// TIA Portal V16 program export: 5 tag tables, 16 data types, 1 data blocks, 21 code blocks (in call order from the OBs), 0 instance data blocks

VAR_GLOBAL   // PLC tag table "Default tag table"
END_VAR

VAR_GLOBAL   // PLC tag table "GLOBAL_CONSTANTS"
END_VAR
VAR_GLOBAL CONSTANT   // user constants
   NUM_AI_RACK : UInt := 1;   // Number of physical analog input points used per rack.
   NUM_DQ_RACK : UInt := 4;   // Number of physical digital output points used per rack.
   NUM_DQ_ROOM : UInt := 9;   // Number of physical digital output points used per room.
   MAX_DQ_PER_ROOM : UInt := 40;   // Max number of physical digital output points per room-based IO module. This needs to equal (NUM_DQ_ROOM + NUM_DQ_RACK*MAX_RACKS_PER_ROOM + EXTRA_DQ_PER_ROOM).
   MAX_VFDS : UInt := 6;   // Total number of VFDs configured in the HW config. This needs to equal MAX_ROOMS * MAX_RACKS_PER_ROOM.
   MAX_ROOMS : UInt := 1;   // Maximum possible number of rooms controlled by a given PLC
   MAX_RACKS_PER_ROOM : UInt := 6;   // Maximum possible number of racks per room
   NUM_AI_ROOM : UInt := 13;   // Number of physical analog input points used per room.
   EXTRA_DQ_PER_ROOM : UInt := 7;   // Number of unused physical digital output points per room-based IO module.
   EXTRA_AI_PER_ROOM : UInt := 1;   // Number of unused physical analog input points per room-based IO module.
   MAX_AI_PER_ROOM : UInt := 20;   // Max number of physical analog input points per room-based IO module. This needs to equal (NUM_AI_ROOM + NUM_AI_RACK*MAX_RACKS_PER_ROOM + EXTRA_AI_PER_ROOM).
END_VAR

VAR_GLOBAL   // PLC tag table "IO"
   GlobalAI AT %I100.0 : "udtArrAIGlobal";   //    {ExternalAccessible false, ExternalVisible false, ExternalWritable false}
   GlobalDQ AT %Q100.0 : "udtArrDQGlobal";   //    {ExternalAccessible false, ExternalVisible false, ExternalWritable false}
END_VAR

VAR_GLOBAL   // PLC tag table "Library Constants"
END_VAR
VAR_GLOBAL CONSTANT   // user constants
   eSTATE_MANUAL : Int := 2;   // State Machine enumeration
   ePBLT_FLASHING_ENABLED : Int := 4;   // HMI PB LT enumeration
   eSTATE_RETRACTING : Int := 5;   // State Machine enumeration
   "IoScaling.S7Analog.Ni100.rScaledMax" : Real := 250.0;
   "IoScaling.S7Analog.Ni100.Climate.rScaledMax" : Real := 250.0;
   eSTEP_StoppingStart : Int := 4000;   // State Machine enumeration
   eSTEP_VerifyCenterComplete : Int := 7999;   // State Machine enumeration
   "IoScaling.S7Analog.150Ohms.rScaledMax" : Real := 150.0;
   "IoScaling.S7Analog.Default.bSwapBytes" : Bool := false;
   eANALOG_INPUTHIGHHIGH : Int := 102;
   eMOTION_DISABLED : Int := 4;   // Status Enumeration - Motion
   "IoScaling.S7Analog.Pt100.iRawMax" : Int := 8500;
   eSTEP_RetractingComplete : Int := 5999;   // State Machine enumeration
   eMODE_MANUAL : Int := 2;   // Mode enumeration
   eANALOG_INPUTINVALID : Int := 101;
   ePBLT_HIDDEN : Int := -1;   // HMI PB LT enumeration
   eVALVE_HOMEON : Int := 6;
   "IoScaling.S7Analog.Pt100.Climate.rScaledMin" : Real := -120.0;
   eHOME_ABS_RET_ABS : Int := 7;   // See MC_Home help for details
   eMOTION_ERROR : Int := 0;   // Status Enumeration - Motion
   ePB_MAINTAINED : Int := 1;   // HMI PB Type enumeration
   LKINCTRL_LENGTH_OF_PATHDATA_NAME : Int := 10;
   LKINCTRL_NO_OF_PATHDATA_ELEMENTS : Int := 15;
   "IoScaling.S7Analog.Pt100.Climate.iRawMax" : Int := 13000;
   eVALVE_ERROR : Int := 2;
   "IoScaling.S7Analog.Types.Pt100.Climate" : Int := 3;
   eMODE_INDEPENDENT : Int := 10;   // Mode
   "IoScaling.S7Analog.600Ohms.rScaledMax" : Real := 600.0;
   eMOTION_RUNNING : Int := 2;   // Status Enumeration - Motion
   "IoScaling.S7Analog.Ni100.Climate.rScaledMin" : Real := -60.0;
   eMOTION_STOPPED : Int := 1;   // Status Enumeration - Motion
   eMOTION_MAINTENANCE : Int := 3;   // Status Enumeration - Motion
   "IoScaling.S7Analog.Ni100.rScaledMin" : Real := -60.0;
   eSTATE_STOPPING : Int := 4;   // State Machine enumeration
   "IoScaling.S7Analog.Pt100.Climate.rScaledMax" : Real := 130.0;
   "IoScaling.S7Analog.Pt100.rScaledMax" : Real := 850.0;
   "IoScaling.S7Analog.Types.Ni100.Climate" : Int := 5;
   ePB_UNLATCH : Int := 3;   // HMI PB Type enumeration
   "IoScaling.S7Analog.Ni100.Climate.iRawMax" : Int := 25000;
   eSTEP_BladeChangeStart : Int := 6000;   // State Machine enumeration
   "IoScaling.S7Analog.300Ohms.rScaledMin" : Real := 0.0;
   "IoScaling.S7Analog.Types.Pt100" : Int := 2;
   LKINCTRL_PI : LReal := 3.1415926535897932846264;
   eVALVE_WORKPOSITION : Int := 3;
   eCAM_SYNCDIRECTION_SHORTESTWAY : Int := 3;   // See MC_CamIn help for details
   "IoScaling.S7Analog.Types.+-V/mA" : Int := 1;
   ePBLT_FLASHING_DISABLED : Int := 5;   // HMI PB LT enumeration
   "IoScaling.S7Analog.150Ohms.rScaledMin" : Real := 0.0;
   eHOME_ACCEPT_CURRENT : Int := 11;   // Used when the configured and current encoders don't match
   LKINCTRL_NO_OF_START_EXECUTE_CMDS : Int := 5;
   ePBLT_TRANSITIONING : Int := 2;   // HMI PB LT enumeration
   SM_ACTIVE_DYNAMICS : Int := 0;
   eVALVE_WORKON : Int := 5;
   "IoScaling.S7Analog.+-V/mA.iRawMax" : Int := 27648;
   eSTATE_INITIALIZATION : Int := 1;   // State Machine enumeration
   LKINCTRL_NO_OF_PATHDATA_PREBUFFER_ELEMENTS : Int := 5;
   eHOME_ABS_RET_OFFSET : Int := 6;   // See MC_Home help for details
   eSTEP_BladeChangeComplete : Int := 6999;   // State Machine enumeration
   eSTEP_RunningComplete : Int := 3999;   // State Machine enumeration
   eANALOG_READY : Int := 100;
   ePBLT_ENABLED : Int := 1;   // HMI PB LT enumeration
   "IoScaling.S7Analog.Pt100.Climate.iRawMin" : Int := -12000;
   eSTATE_RUNNING : Int := 3;   // State Machine enumeration
   LKINCTRL_NO_OF_LAST_FLAG : Int := 15;
   "IoScaling.S7Analog.Ni100.iRawMax" : Int := 2500;
   "IoScaling.S7Analog.Types.Default" : Int := 0;
   eHOME_ACCEPT_CONFIG : Int := 12;   // Used when the configured and current encoders don't match
   eSTEP_RunningStart : Int := 3000;   // State Machine enumeration
   "IoScaling.S7Analog.Default.iRawMin" : Int := 0;
   ePBLT_ACTIVE : Int := 3;   // HMI PB LT enumeration
   "IoScaling.S7Analog.Types.Ni100" : Int := 4;
   eMODE_AUTO : Int := 1;   // Mode enumeration
   "IoScaling.S7Analog.Default.iRawMax" : Int := 27648;
   ePBLT_DISABLED : Int := 0;   // HMI PB LT enumeration
   LKINCTRL_NO_OF_SEQ_EXECUTE_CMDS : Int := 5;
   eSTEP_StoppingComplete : Int := 4999;   // State Machine enumeration
   "IoScaling.S7Analog.Ni100.Climate.iRawMin" : Int := -6000;
   "IoScaling.S7Analog.Pt100.iRawMin" : Int := -2000;
   ePB_LATCH : Int := 2;   // HMI PB Type enumeration
   eVALVE_ESTOP : Int := 1;
   eSTEP_RetractingStart : Int := 5000;   // State Machine enumeration
   "IoScaling.S7Analog.300Ohms.rScaledMax" : Real := 300.0;
   eANALOG_INPUTLOW : Int := 105;
   "IoScaling.S7Analog.Pt100.rScaledMin" : Real := -200.0;
   eSTATE_BLADECHANGE : Int := 6;   // State Machine enumeration
   "IoScaling.S7Analog.600Ohms.rScaledMin" : Real := 0.0;
   eSTATE_VERIFYCENTER : Int := 7;   // State Machine enumeration
   eVALVE_STOPPED : Int := 0;
   eCAM_SYNCPROFILEREFERENCE_LEADINGVALUEDISTANCE : Int := 1;   // See MC_CamIn help for details
   "IoScaling.S7Analog.Ni100.iRawMin" : Int := -600;
   ePB_HELD : Int := 4;   // HMI PB Type enumeration
   LKINCTRL_NO_OF_CMD_SETFLAGS : Int := 8;
   eSTEP_VerifyCenterStart : Int := 7000;   // State Machine enumeration
   eVALVE_HOMEPOSITION : Int := 4;
   eANALOG_INPUTHIGH : Int := 104;
   eANALOG_INPUTLOWLOW : Int := 103;
   "IoScaling.S7Analog.+-V/mA.iRawMin" : Int := -27648;
   ePB_MOMENTARY : Int := 0;   // HMI PB Type enumeration
   "Modes.PID.Pretuning" : Int := 1;
   "TotalizerTimeUnits.DAYS" : Int := 4;
   "HMI.Status.ForwardWork" : Int := 3;
   "FIFO.iQueueDisabled" : Int := -1;
   "Handshakes.iSize" : Int := 5;
   "Modes.Auto" : Int := 1;
   "HMI.Status.Generic1" : Int := 101;
   "Simocode.Types.DirectStarter" : Int := 1;
   "Estop.MinSetPoint" : Int := 0;
   "Simocode.Types.OverloadRelay" : Int := 0;
   "HMI.Status.SimulatedReverseHome" : Int := 8;
   "TotalizerTimeUnits.MILLISECONDS" : Int := 0;
   "HMI.Status.Generic4" : Int := 104;
   "SoftStarter.HMI.Status.EStop" : Int := 1;
   "HMI.Status.OnForwardWork" : Int := 5;
   "DataTypes.iMaxInt" : Int := 32767;
   "FIFO.iQueueSize" : Int := 5;
   "Modes.PID.ManualMode" : Int := 4;
   "TotalizerTimeUnits.SECONDS" : Int := 1;
   "SoftStarter.Types.3RW30" : Int := 30;
   "HMI.Status.Generic3" : Int := 103;
   "HMI.Status.OnReverseHome" : Int := 6;
   "HMI.Status.Estop" : Int := 1;
   "SoftStarter.HMI.Status.Error" : Int := 2;
   "HMI.Status.Generic6" : Int := 106;
   "DataTypes.rMaxReal" : Real := 3.402823e38;
   "SoftStarter.HMI.Status.Off" : Int := 0;
   "Modes.PID.Inactive" : Int := 0;
   "HMI.Status.GenericNone" : Int := 100;
   "HMI.Status.Generic2" : Int := 102;
   "Modes.PID.AutoMode" : Int := 3;
   "SoftStarter.HMI.Status.On" : Int := 4;
   "Estop.HMISetPoint" : Int := 2;
   "HMI.Status.ReverseHome" : Int := 4;
   "DataTypes.rMinReal" : Real := -3.402823e38;
   "TotalizerTimeUnits.MINUTES" : Int := 2;
   "Modes.PID.FineTuning" : Int := 2;
   "TotalizerTimeUnits.HOURS" : Int := 3;
   "Ramp.Timed" : Int := 1;
   "Estop.MaxSetPoint" : Int := 1;
   "SoftStarter.Types.3RW40" : Int := 40;
   "Ramp.Continuous" : Int := 0;
   "HMI.Status.Generic5" : Int := 105;
   "Modes.Manual" : Int := 2;
   "Modes.Stop" : Int := 0;
   "HMI.Status.SimulatedOnReverseHome" : Int := 10;
   "Simocode.Types.ReversingStarter" : Int := 2;
   "Modes.Independent" : Int := 10;
   "DataTypes.iMinInt" : Int := -32768;
   "SoftStarter.HMI.Status.RampUp" : Int := 3;
   "SoftStarter.HMI.Status.RampDown" : Int := 5;
   "HMI.Status.Error" : Int := 2;
   "HMI.Status.SimulatedOnForwardWork" : Int := 9;
   "HMI.Status.SimulatedForwardWork" : Int := 7;
   "HMI.Status.Stopped" : Int := 0;
END_VAR

VAR_GLOBAL   // PLC tag table "System Bits"
   System_Byte AT %MB1 : Byte;   //    {ExternalAccessible false, ExternalVisible false, ExternalWritable false}
   AlwaysFALSE AT %M1.3 : Bool;   //    {ExternalAccessible false, ExternalVisible false, ExternalWritable false}
   "Clock_1.25Hz" AT %M0.4 : Bool;   //    {ExternalAccessible false, ExternalVisible false, ExternalWritable false}
   Clock_1Hz AT %M0.5 : Bool;   //    {ExternalAccessible false, ExternalVisible false, ExternalWritable false}
   "Clock_0.5Hz" AT %M0.7 : Bool;   //    {ExternalAccessible false, ExternalVisible false, ExternalWritable false}
   FirstScan AT %M1.0 : Bool;   //    {ExternalAccessible false, ExternalVisible false, ExternalWritable false}
   Clock_Byte AT %MB0 : Byte;   //    {ExternalAccessible false, ExternalVisible false, ExternalWritable false}
   "Clock_2.5Hz" AT %M0.2 : Bool;   //    {ExternalAccessible false, ExternalVisible false, ExternalWritable false}
   "Clock_0.625Hz" AT %M0.6 : Bool;   //    {ExternalAccessible false, ExternalVisible false, ExternalWritable false}
   Clock_5Hz AT %M0.1 : Bool;   //    {ExternalAccessible false, ExternalVisible false, ExternalWritable false}
   Clock_10Hz AT %M0.0 : Bool;   //    {ExternalAccessible false, ExternalVisible false, ExternalWritable false}
   AlwaysTRUE AT %M1.2 : Bool;   //    {ExternalAccessible false, ExternalVisible false, ExternalWritable false}
   DiagStatusUpdate AT %M1.1 : Bool;   //    {ExternalAccessible false, ExternalVisible false, ExternalWritable false}
   Clock_2Hz AT %M0.3 : Bool;   //    {ExternalAccessible false, ExternalVisible false, ExternalWritable false}
END_VAR

TYPE "udtFertigationSettings"
VERSION : 0.1
   STRUCT
      tMeasurementTime { ExternalAccessible := 'False'; ExternalVisible := 'False'; ExternalWritable := 'False'} : Time;   // Duration of cycle through M loop before measurement taken (s)
      rMeasurementVolume { ExternalAccessible := 'False'; ExternalVisible := 'False'; ExternalWritable := 'False'} : Real;   // Amount of water to receive from rack for measurement (L)
      bNutrientAEnable { ExternalAccessible := 'False'; ExternalVisible := 'False'; ExternalWritable := 'False'} : Bool;   // Enables nutrient A for use in dosing
      bNutrientBEnable { ExternalAccessible := 'False'; ExternalVisible := 'False'; ExternalWritable := 'False'} : Bool;   // Enables nutrient B for use in dosing
      rISELowSP { ExternalAccessible := 'False'; ExternalVisible := 'False'; ExternalWritable := 'False'} : Real;   // Low setpoint for ISE measurement for dosing
      rISEHighSP { ExternalAccessible := 'False'; ExternalVisible := 'False'; ExternalWritable := 'False'} : Real;   // High setpoint for ISE measurement for dosing
      tNutrientDosingDuration { ExternalAccessible := 'False'; ExternalVisible := 'False'; ExternalWritable := 'False'} : Time;   // Duration for which to add a nutrient during dosing (s)
      bDosingActive { ExternalAccessible := 'False'; ExternalVisible := 'False'; ExternalWritable := 'False'} : Bool;   // Rack was dosed on last MD cycle and is below high SP
      rOperatingVolume { ExternalAccessible := 'False'; ExternalVisible := 'False'; ExternalWritable := 'False'} : Real;   // Operating volume for fill after dosing (L)
      rTotalShelfVolume { ExternalAccessible := 'False'; ExternalVisible := 'False'; ExternalWritable := 'False'} : Real;
      rMaxReservoirVolume { ExternalAccessible := 'False'; ExternalVisible := 'False'; ExternalWritable := 'False'} : Real;   // Maximum water capacity of the rack (L)
      rMinReservoirVolume { ExternalAccessible := 'False'; ExternalVisible := 'False'; ExternalWritable := 'False'} : Real;   // Minimum water capacity of the rack (L)
      rRackCurrentVolume { ExternalAccessible := 'False'; ExternalVisible := 'False'; ExternalWritable := 'False'} : Real;   // Current rack fill level (L)
      bPumpAtStandstill { ExternalAccessible := 'False'; ExternalVisible := 'False'; ExternalWritable := 'False'} : Bool;
      bEndDischargeCommand { ExternalAccessible := 'False'; ExternalVisible := 'False'; ExternalWritable := 'False'} : Bool;
      tDischargeTime { ExternalAccessible := 'False'; ExternalVisible := 'False'; ExternalWritable := 'False'} : Time;
      bEnableIncomingRotate { ExternalAccessible := 'False'; ExternalVisible := 'False'; ExternalWritable := 'False'} : Bool;   // Rack is in M&D mode and circulating state
   END_STRUCT;

END_TYPE

TYPE "udtModbusValBool"
VERSION : 0.1
   STRUCT
      iAddr { ExternalAccessible := 'False'; ExternalVisible := 'False'; ExternalWritable := 'False'} : UInt;   // Full modbus address (1 indexed, including offset for object type)
      bVal { ExternalAccessible := 'False'; ExternalVisible := 'False'; ExternalWritable := 'False'} : Bool;
   END_STRUCT;

END_TYPE

TYPE "udtModbusValReal"
VERSION : 0.1
   STRUCT
      iRegister { ExternalAccessible := 'False'; ExternalVisible := 'False'; ExternalWritable := 'False'} : UInt;   // Full modbus address (1 indexed, including offset for object type)
      rVal { ExternalAccessible := 'False'; ExternalVisible := 'False'; ExternalWritable := 'False'} : Real;
   END_STRUCT;

END_TYPE

TYPE "udtNutrientReading"
VERSION : 0.1
   STRUCT
      rISEReading { ExternalVisible := 'False'; ExternalWritable := 'False'} : Real;   // Nutrient measurement level
      rORPReading { ExternalVisible := 'False'; ExternalWritable := 'False'} : Real;   // Nutrient measurement level
      rECReading { ExternalVisible := 'False'; ExternalWritable := 'False'} : Real;   // Nutrient measurement level
      rpHReading { ExternalVisible := 'False'; ExternalWritable := 'False'} : Real;   // Nutrient measurement level
   END_STRUCT;

END_TYPE

TYPE "udtTimeOfDaySetpoint"
VERSION : 0.1
   STRUCT
      TimeOfDaySeconds { ExternalVisible := 'False'} : DInt := -1;   // -1 default for unused setpoint
      rSetpoint { ExternalVisible := 'False'} : Real;
   END_STRUCT;

END_TYPE

TYPE "udtArrAIGlobal"
VERSION : 0.1
   STRUCT
      Room { ExternalAccessible := 'False'; ExternalVisible := 'False'; ExternalWritable := 'False'; S7_SetPoint := 'False'} : Array[1.."MAX_ROOMS"] of "udtArrAIRoom";
   END_STRUCT;

END_TYPE

TYPE "udtArrAIRoom"
VERSION : 0.1
   STRUCT
      AI { ExternalAccessible := 'False'; ExternalVisible := 'False'; ExternalWritable := 'False'} : Array[1.."MAX_AI_PER_ROOM"] of Int;
   END_STRUCT;

END_TYPE

TYPE "udtArrDQGlobal"
VERSION : 0.1
   STRUCT
      Room { ExternalAccessible := 'False'; ExternalVisible := 'False'; ExternalWritable := 'False'; S7_SetPoint := 'False'} : Array[1.."MAX_ROOMS"] of "udtArrDQRoom";
   END_STRUCT;

END_TYPE

TYPE "udtArrDQRoom"
VERSION : 0.1
   STRUCT
      DQ { ExternalAccessible := 'False'; ExternalVisible := 'False'; ExternalWritable := 'False'} : Array[1.."MAX_DQ_PER_ROOM"] of Bool;
   END_STRUCT;

END_TYPE

TYPE "udtDigitalOutput"
VERSION : 0.1
   STRUCT
      bAutoVal { ExternalVisible := 'False'; ExternalWritable := 'False'} : Bool;   // Value set by the program
      bOverrideVal { ExternalVisible := 'False'} : Bool;   // Value set by the user, tracks bAuto when bOverrideEnable=0
      bStatus { ExternalVisible := 'False'; ExternalWritable := 'False'} : Bool;   // Value being written to actual output
      bOverrideEnable { ExternalVisible := 'False'} : Bool;   // Sets bOut to bOverride
   END_STRUCT;

END_TYPE

TYPE "udtRackAI"
VERSION : 0.1
   STRUCT
      IW_ReservoirLevel { ExternalAccessible := 'False'; ExternalVisible := 'False'; ExternalWritable := 'False'} : Int;
   END_STRUCT;

END_TYPE

TYPE "udtRackDQ"
VERSION : 0.1
   STRUCT
      Q_SupplySolenoid { ExternalAccessible := 'False'; ExternalVisible := 'False'; ExternalWritable := 'False'} : Bool;
      Q_ReturnSolenoid { ExternalAccessible := 'False'; ExternalVisible := 'False'; ExternalWritable := 'False'} : Bool;
      Q_ShelfSolenoid { ExternalAccessible := 'False'; ExternalVisible := 'False'; ExternalWritable := 'False'} : Bool;
      Q_Lights { ExternalAccessible := 'False'; ExternalVisible := 'False'; ExternalWritable := 'False'} : Bool;
   END_STRUCT;

END_TYPE

TYPE "udtRoomAI"
VERSION : 0.1
   STRUCT
      IW_RoomTemperature_1 { ExternalAccessible := 'False'; ExternalVisible := 'False'; ExternalWritable := 'False'} : Int;
      IW_RoomTemperature_2 { ExternalAccessible := 'False'; ExternalVisible := 'False'; ExternalWritable := 'False'} : Int;
      IW_RoomHumidity_1 { ExternalAccessible := 'False'; ExternalVisible := 'False'; ExternalWritable := 'False'} : Int;
      IW_RoomHumidity_2 { ExternalAccessible := 'False'; ExternalVisible := 'False'; ExternalWritable := 'False'} : Int;
      IW_TankLevel { ExternalAccessible := 'False'; ExternalVisible := 'False'; ExternalWritable := 'False'} : Int;
      IW_NutrientALevel { ExternalAccessible := 'False'; ExternalVisible := 'False'; ExternalWritable := 'False'} : Int;
      IW_NutrientBLevel { ExternalAccessible := 'False'; ExternalVisible := 'False'; ExternalWritable := 'False'} : Int;
      IW_NutrientAcidLevel { ExternalAccessible := 'False'; ExternalVisible := 'False'; ExternalWritable := 'False'} : Int;
      IW_pHSensor { ExternalAccessible := 'False'; ExternalVisible := 'False'; ExternalWritable := 'False'} : Int;
      IW_ECSensor { ExternalAccessible := 'False'; ExternalVisible := 'False'; ExternalWritable := 'False'} : Int;
      IW_ISESensor { ExternalAccessible := 'False'; ExternalVisible := 'False'; ExternalWritable := 'False'} : Int;
      IW_ORPSensor { ExternalAccessible := 'False'; ExternalVisible := 'False'; ExternalWritable := 'False'} : Int;
      IW_CO2Sensor { ExternalAccessible := 'False'; ExternalVisible := 'False'; ExternalWritable := 'False'} : Int;
   END_STRUCT;

END_TYPE

TYPE "udtRoomDQ"
VERSION : 0.1
   STRUCT
      Q_MPathSolenoid { ExternalAccessible := 'False'; ExternalVisible := 'False'; ExternalWritable := 'False'} : Bool;
      Q_FreshWaterSolenoid { ExternalAccessible := 'False'; ExternalVisible := 'False'; ExternalWritable := 'False'} : Bool;
      Q_DischargeSolenoid { ExternalAccessible := 'False'; ExternalVisible := 'False'; ExternalWritable := 'False'} : Bool;
      Q_TankReturnSolenoid { ExternalAccessible := 'False'; ExternalVisible := 'False'; ExternalWritable := 'False'} : Bool;
      Q_NutrientAEnable { ExternalAccessible := 'False'; ExternalVisible := 'False'; ExternalWritable := 'False'} : Bool;
      Q_NutrientBEnable { ExternalAccessible := 'False'; ExternalVisible := 'False'; ExternalWritable := 'False'} : Bool;
      Q_NutrientAcidEnable { ExternalAccessible := 'False'; ExternalVisible := 'False'; ExternalWritable := 'False'} : Bool;
      Q_NutrientMixingPumps { ExternalAccessible := 'False'; ExternalVisible := 'False'; ExternalWritable := 'False'} : Bool;
      Q_CO2Solenoid { ExternalAccessible := 'False'; ExternalVisible := 'False'; ExternalWritable := 'False'} : Bool;
   END_STRUCT;

END_TYPE

TYPE "udtError_VFD"
VERSION : 0.1
   STRUCT
      MotorProtectorTripped { ExternalWritable := 'False'} : Bool;   // Motor protector tripped
      LocalDisconnectOff { ExternalWritable := 'False'} : Bool;   // Motor disconnect off
      ClutchTripped { ExternalWritable := 'False'} : Bool;   // Clutch tripped
      NoContactorFeedback { ExternalWritable := 'False'} : Bool;   // No feedback from motor contactor
      ContactorStillOn { ExternalWritable := 'False'} : Bool;   // Contactor still on
      NoSignalForward { ExternalWritable := 'False'} : Bool;   // No signal forward from VFD
      NoSignalReverse { ExternalWritable := 'False'} : Bool;   // No signal reverse from VFD
      MotorNotStopped { ExternalWritable := 'False'} : Bool;   // Motor doesn't stop
      MaxFrequencyReached { ExternalWritable := 'False'} : Bool;   // Max frequency reached
      Overcurrent { ExternalWritable := 'False'} : Bool;   // VFD overcurrent
      MotorOverload { ExternalWritable := 'False'} : Bool;   // Motor overload
      VFDOverload { ExternalWritable := 'False'} : Bool;   // VFD overload
      GeneralFault { ExternalWritable := 'False'} : Bool;   // VFD fault
      NoCoolingFanFeedback { ExternalWritable := 'False'} : Bool;   // No feedback from cooling fan
   END_STRUCT;

END_TYPE

TYPE "udtHMI_VFD_Control"
VERSION : 0.1
   STRUCT
      iMode : Int;   // Current mode
      iErrorCode { ExternalWritable := 'False'} : Int;   // Error code
      iStatus { ExternalWritable := 'False'} : Int;   // Status for HMI display
      rManualSpeedSP { S7_SetPoint := 'True'} : Real;   // Speed set point for manual mode
      rAutoSpeedSP { ExternalWritable := 'False'} : Real;   // Speed set point for automatic mode
      rActualSpeed { ExternalWritable := 'False'} : Real;   // Actual motor speed
      rActualCurrent { ExternalWritable := 'False'} : Real;   // Actual motor current
      rActualPower { ExternalWritable := 'False'} : Real;   // Actual motor power
      bPB_ResetError : Bool;   // PB Reset errors
      bPB_Forward : Bool;   // PB Move forward in manual mode
      bPB_Reverse : Bool;   // PB Move reverse in manual mode
      bPB_Stop : Bool;   // PB Stop in manual mode
      bPBEN_ResetError { ExternalWritable := 'False'} : Bool;   // PB Reset errors enabled
      bPBEN_Forward { ExternalWritable := 'False'} : Bool;   // PB Forward enabled
      bPBEN_Reverse { ExternalWritable := 'False'} : Bool;   // PB Reverse enabled
      bPBEN_Stop { ExternalWritable := 'False'} : Bool;   // PB Stop enabled
      bForwardOn { ExternalWritable := 'False'} : Bool;   // Moving forward
      bReverseOn { ExternalWritable := 'False'} : Bool;   // Moving Reverse
      bSignalForward { ExternalWritable := 'False'} : Bool;   // Forward signal
      bSignalReverse { ExternalWritable := 'False'} : Bool;   // Reverse signal
      bError { ExternalWritable := 'False'} : Bool;   // Overall error
      bInterlock { ExternalWritable := 'False'} : Bool;   // VFD Interlocked
   END_STRUCT;

END_TYPE

DATA_BLOCK "dbMain"
{ S7_Optimized_Access := 'TRUE' }
VERSION : 0.1
NON_RETAIN
"fbMain"

BEGIN
   Room[1].Fertigation.Controls.rTankEmptyLevel := 60.0;
   Room[1].AI_ISESensor.Config.rHighCalibration := 900.0;

END_DATA_BLOCK

ORGANIZATION_BLOCK "Main"   // OB1, LAD, ProgramCycle
TITLE = "Main Program Sweep (Cycle)"
{ S7_Optimized_Access := 'TRUE' }
VERSION : 0.1
// stored: AutoNumber true, IsIECCheckEnabled false, SetENOAutomatically false
   VAR_INPUT
      Initial_Call : Bool;   // Initial call of this OB
      Remanence : Bool;   // =True, if remanent data are available
   END_VAR
BEGIN

REGION Network 1
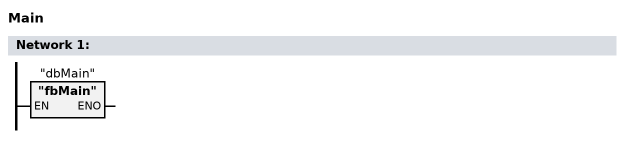
   RUNG wire#powerrail
      "dbMain"()
   END_RUNG
   // the same network as SCL:
   "dbMain"();   // "fbMain"
END_REGION
END_ORGANIZATION_BLOCK

FUNCTION_BLOCK "fbMain"   // FB4, LAD
{ S7_Optimized_Access := 'TRUE' }
VERSION : 0.1
// Main block which calls all room FBs and holds all parameters in instance memory.
// stored: AutoNumber true, IsIECCheckEnabled false, IsRetainMemResEnabled false, MemoryReserve 100, SetENOAutomatically false, UDAEnableTagReadback false
   VAR
      Room { ExternalVisible := 'False'} : Array[1.."MAX_ROOMS"] of "fbRoom";
      Config { ExternalVisible := 'False'} : "fbConfig";
   END_VAR
   VAR_TEMP
      iRoomCount : Int;
      iRackCount : Int;
      iPos : DInt;
   END_VAR
BEGIN

REGION Network 1 (SCL): Call config FB
   // bInSimulation := TRUE skips IO device configuration steps
   #Config(bInSimulation := #Config.bInSimulation);
END_REGION

REGION Network 2 (SCL): Map input array to all room and rack inputs
   IF #Config.Status.bDone THEN

       FOR #iRoomCount := 1 TO UINT_TO_INT("MAX_ROOMS") DO

           #iPos := 1; // input array is 1 indexed

           MOVE_BLK(IN := "GlobalAI".Room[#iRoomCount].AI[#iPos],
                    COUNT := "NUM_AI_ROOM",
                    OUT => #Room[#iRoomCount].arrAI[1]);

           #iPos += "NUM_AI_ROOM";


           FOR #iRackCount := 1 TO UINT_TO_INT("MAX_RACKS_PER_ROOM") DO

               MOVE_BLK(IN := "GlobalAI".Room[#iRoomCount].AI[#iPos],
                        COUNT := "NUM_AI_RACK",
                        OUT => #Room[#iRoomCount].Rack[#iRackCount].arrAI[1]);

               #iPos += "NUM_AI_RACK";

           END_FOR;

           #iPos += "EXTRA_AI_PER_ROOM"; // skip over unused points

       END_FOR;

   END_IF;
END_REGION

REGION Network 3 (SCL): TEMPORARY- Remap inputs from temporary IO tag table
   #Room[1].arrAI[1] := "IW_RoomTemperature_1";
   #Room[1].arrAI[2] := "IW_RoomTemperature_2";
   #Room[1].arrAI[3] := "IW_RoomHumidity_1";
   #Room[1].arrAI[4] := "IW_RoomHumidity_2";
   #Room[1].arrAI[5] := "IW_TankLevel";
   #Room[1].arrAI[6] := "IW_NutrientALevel";
   #Room[1].arrAI[7] := "IW_NutrientBLevel";
   #Room[1].arrAI[8] := "IW_NutrientAcidLevel";
   #Room[1].arrAI[9] := "IW_pHSensor";
   #Room[1].arrAI[10] := "IW_ECSensor";
   #Room[1].arrAI[11] := "IW_ISESensor";
   #Room[1].arrAI[12] := "IW_ORPSensor";
   #Room[1].arrAI[13] := "IW_CO2Sensor";

   #Room[1].Rack[1].arrAI[1] := "IW_Rack1Level";
   #Room[1].Rack[2].arrAI[1] := "IW_Rack2Level";
   #Room[1].Rack[3].arrAI[1] := "IW_Rack3Level";
   #Room[1].Rack[4].arrAI[1] := "IW_Rack4Level";
   #Room[1].Rack[5].arrAI[1] := "IW_Rack5Level";
   #Room[1].Rack[6].arrAI[1] := "IW_Rack6Level";
END_REGION

REGION Network 4 (SCL): Call FBs for all configured rooms
   IF #Config.Status.bDone THEN

       FOR #iRoomCount := 1 TO #Config.iNumRooms DO

           #Room[#iRoomCount](arrAI := #Room[#iRoomCount].arrAI,
                              arrDQ=> #Room[#iRoomCount].arrDQ);

       END_FOR;

   END_IF;
END_REGION

REGION Network 5 (SCL): Combine all room and rack outputs into a single output array
   IF #Config.Status.bDone THEN

       FOR #iRoomCount := 1 TO UINT_TO_INT("MAX_ROOMS") DO

           #iPos := 1; // output array is 1 indexed

           MOVE_BLK(IN := #Room[#iRoomCount].arrDQ[1],
                    COUNT := "NUM_DQ_ROOM",
                    OUT => "GlobalDQ".Room[#iRoomCount].DQ[#iPos]);

           #iPos += "NUM_DQ_ROOM";


           FOR #iRackCount := 1 TO UINT_TO_INT("MAX_RACKS_PER_ROOM") DO

               MOVE_BLK(IN := #Room[#iRoomCount].Rack[#iRackCount].arrDQ[1],
                        COUNT := "NUM_DQ_RACK",
                        OUT => "GlobalDQ".Room[#iRoomCount].DQ[#iPos]);

               #iPos += "NUM_DQ_RACK";

           END_FOR;

           #iPos += "EXTRA_DQ_PER_ROOM"; // skip over unused points

       END_FOR;

   END_IF;
END_REGION

REGION Network 6 (SCL): TEMPORARY- Remap inputs to temporary IO tag table
   "Q_MPathSolenoid" := #Room[1].arrDQ[1];
   "Q_FreshWaterSolenoid" := #Room[1].arrDQ[2];
   "Q_DischargeSolenoid" := #Room[1].arrDQ[3];
   "Q_TankReturnSolenoid" := #Room[1].arrDQ[4];
   "Q_NutrientAEnable" := #Room[1].arrDQ[5];
   "Q_NutrientBEnable" := #Room[1].arrDQ[6];
   "Q_NutrientAcidEnable" := #Room[1].arrDQ[7];
   "Q_NutrientMixingPumps" := #Room[1].arrDQ[8];
   "Q_CO2Solenoid" := #Room[1].arrDQ[9];

   "Q_Rack1Supply" := #Room[1].Rack[1].arrDQ[1];
   "Q_Rack1Return" := #Room[1].Rack[1].arrDQ[2];
   "Q_Rack1Shelves" := #Room[1].Rack[1].arrDQ[3];
   "Q_Rack1Lights" := #Room[1].Rack[1].arrDQ[4];
   "Q_Rack2Supply" := #Room[1].Rack[2].arrDQ[1];
   "Q_Rack2Return" := #Room[1].Rack[2].arrDQ[2];
   "Q_Rack2Shelves" := #Room[1].Rack[2].arrDQ[3];
   "Q_Rack2Lights" := #Room[1].Rack[2].arrDQ[4];
   "Q_Rack3Supply" := #Room[1].Rack[3].arrDQ[1];
   "Q_Rack3Return" := #Room[1].Rack[3].arrDQ[2];
   "Q_Rack3Shelves" := #Room[1].Rack[3].arrDQ[3];
   "Q_Rack3Lights" := #Room[1].Rack[3].arrDQ[4];
   "Q_Rack4Supply" := #Room[1].Rack[4].arrDQ[1];
   "Q_Rack4Return" := #Room[1].Rack[4].arrDQ[2];
   "Q_Rack4Shelves" := #Room[1].Rack[4].arrDQ[3];
   "Q_Rack4Lights" := #Room[1].Rack[4].arrDQ[4];
   "Q_Rack5Supply" := #Room[1].Rack[5].arrDQ[1];
   "Q_Rack5Return" := #Room[1].Rack[5].arrDQ[2];
   "Q_Rack5Shelves" := #Room[1].Rack[5].arrDQ[3];
   "Q_Rack5Lights" := #Room[1].Rack[5].arrDQ[4];
   "Q_Rack6Supply" := #Room[1].Rack[6].arrDQ[1];
   "Q_Rack6Return" := #Room[1].Rack[6].arrDQ[2];
   "Q_Rack6Shelves" := #Room[1].Rack[6].arrDQ[3];
   "Q_Rack6Lights" := #Room[1].Rack[6].arrDQ[4];
END_REGION
END_FUNCTION_BLOCK

FUNCTION_BLOCK "fbConfig"
{ S7_Optimized_Access := 'TRUE' }
VERSION : 0.1
   VAR_INPUT RETAIN
      bInSimulation { ExternalAccessible := 'False'; ExternalVisible := 'False'; ExternalWritable := 'False'} : Bool := false;   // If true, skips IO reconfig steps
   END_VAR

   VAR RETAIN
      Controls { ExternalVisible := 'False'} : Struct
         iSetNumRooms { ExternalVisible := 'False'} : Int := 1;
         arrSetNumRacksPerRoom { ExternalVisible := 'False'} : Array[1.."MAX_ROOMS"] of Int := [6];
         bSetConfig { ExternalVisible := 'False'} : Bool := false;
      END_STRUCT;
   END_VAR
   VAR 
      Status { ExternalVisible := 'False'; ExternalWritable := 'False'} : Struct
         bDone { ExternalVisible := 'False'; ExternalWritable := 'False'} : Bool;
         bBusy { ExternalVisible := 'False'; ExternalWritable := 'False'} : Bool;
         bError { ExternalVisible := 'False'; ExternalWritable := 'False'} : Bool;
         ErrorMsg { ExternalVisible := 'False'; ExternalWritable := 'False'} : String;
      END_STRUCT;
      iNumRooms { ExternalVisible := 'False'; ExternalWritable := 'False'} : Int := 0;
      iStep { ExternalAccessible := 'False'; ExternalVisible := 'False'; ExternalWritable := 'False'} : Int;
      iNextStep { ExternalAccessible := 'False'; ExternalVisible := 'False'; ExternalWritable := 'False'} : Int;
      R_TRIG_SetConfig {InstructionName := 'R_TRIG'; LibVersion := '1.0'; ExternalAccessible := 'False'; ExternalVisible := 'False'; ExternalWritable := 'False'} : R_TRIG;
      ReconfigIOSystem {InstructionName := 'ReconfigIOSystem'; LibVersion := '1.2'; ExternalAccessible := 'False'; ExternalVisible := 'False'; ExternalWritable := 'False'; S7_SetPoint := 'False'} : ReconfigIOSystem;
      arrVfdDeviceConfig { ExternalAccessible := 'False'; ExternalVisible := 'False'; ExternalWritable := 'False'} : Array[-2.."MAX_VFDS"] of Word;
   END_VAR

   VAR_TEMP 
      iRoomIndex : Int;
      iRackIndex : Int;
      arrTelegrams : Array[1.."MAX_VFDS"] of HW_SUBMODULE;
      arrIoDeviceIds : Array[1.."MAX_VFDS"] of HW_DEVICE;
      i : Int;
      iVfdCount : Int;
      bSettingsValid : Bool;
      strErrorCode : String;
      retVal : Word;
   END_VAR

   VAR CONSTANT 
      eStep_ValidateConfig : Int;
      eStep_SetUp : Int := 1;
      eStep_Deactivate : Int := 2;
      eStep_WaitForDeactivate : Int := 3;
      eStep_Reconfig : Int := 4;
      eStep_WaitForReconfig : Int := 5;
      eStep_Restart : Int := 6;
      eStep_Done : Int := 7;
      eStep_Error : Int := 8;
   END_VAR


BEGIN
	// Enables VFDs and IO racks based on the number of configured rooms and racks.
	// The intention is for everything to be configurable via the OPC UA interface and nothing
	// needs to be changed in TIA Portal, so that all deployments regardless of size can use the same codebase.
	
	// Global constants for reference:
	(*
	"MAX_ROOMS"
	"MAX_RACKS_PER_ROOM"
	"MAX_VFDS"
	
	"NUM_AI_ROOM"
	"NUM_AI_RACK"
	"MAX_AI_TOTAL"
	
	"NUM_DQ_ROOM"
	"NUM_DQ_RACK"
	"MAX_DQ_TOTAL"
	*)
	
	REGION 0: Validate config, set num racks and rooms
	    
	    // wait for start command
	    #R_TRIG_SetConfig(CLK:= #Controls.bSetConfig);
	    
	    // also trigger on PLC startup
	    IF "FirstScan" OR #iStep = #eStep_ValidateConfig OR
	        (#R_TRIG_SetConfig.Q AND (#iStep = #eStep_Done OR #iStep = #eStep_Error) ) THEN
	        
	        REGION Check error conditions            
	            // make sure specified number of rooms and racks is valid
	            #bSettingsValid := TRUE;
	            #Status.ErrorMsg := '';
	            
	            IF "MAX_VFDS" <> "MAX_ROOMS" * "MAX_RACKS_PER_ROOM" THEN
	                #bSettingsValid := FALSE;
	                #Status.ErrorMsg := CONCAT(IN1 := #Status.ErrorMsg, IN2 := ' MAX_VFDS != MAX_ROOMS*MAX_RACKS ');
	            END_IF;
	            
	            IF #Controls.iSetNumRooms > "MAX_ROOMS" THEN
	                #bSettingsValid := FALSE;
	                #Status.ErrorMsg := CONCAT(IN1 := #Status.ErrorMsg, IN2 := ' NumRooms > MAX ');
	            END_IF;
	            
	            FOR #i := 1 TO UINT_TO_INT("MAX_ROOMS") DO
	                IF #Controls.arrSetNumRacksPerRoom[#i] > "MAX_RACKS_PER_ROOM" THEN
	                    #bSettingsValid := FALSE;
	                    #Status.ErrorMsg := CONCAT(IN1 := #Status.ErrorMsg, IN2 := ' NumRacks > MAX ');
	                    EXIT;
	                END_IF;
	            END_FOR;
	            
	            IF "MAX_AI_PER_ROOM" <> ("NUM_AI_ROOM" + "NUM_AI_RACK" * "MAX_RACKS_PER_ROOM" + "EXTRA_AI_PER_ROOM") OR ( "MAX_AI_PER_ROOM" MOD 4 <> 0) THEN
	                #bSettingsValid := FALSE;
	                #Status.ErrorMsg := CONCAT(IN1 := #Status.ErrorMsg, IN2 := ' MAX_AI_PER_ROOM incorrect ');
	            END_IF;
	            
	            IF "MAX_DQ_PER_ROOM" <> ("NUM_DQ_ROOM" + "NUM_DQ_RACK" * "MAX_RACKS_PER_ROOM" + "EXTRA_DQ_PER_ROOM") OR ( "MAX_DQ_PER_ROOM" MOD 8 <> 0) THEN
	                #bSettingsValid := FALSE;
	                #Status.ErrorMsg := CONCAT(IN1 := #Status.ErrorMsg, IN2 := ' MAX_DQ_PER_ROOM incorrect ');
	            END_IF;
	            
	        END_REGION
	        
	        IF #bSettingsValid THEN
	            // set number of rooms
	            #iNumRooms := #Controls.iSetNumRooms;
	            
	            FOR #iRoomIndex := 1 TO #iNumRooms DO
	                // set number of racks in each room
	                "dbMain".Room[#iRoomIndex].Config.iNumRacks := #Controls.arrSetNumRacksPerRoom[#iRoomIndex];
	            END_FOR;
	            
	            #iNextStep := #eStep_SetUp;
	            
	        ELSE
	            #iNextStep := #eStep_Error;
	            
	        END_IF;
	        
	    END_IF;
	    
	END_REGION
	
	REGION 1: Set up params
	    
	    IF #iStep = #eStep_SetUp THEN
	        
	        REGION Map VFD IO device system constants
	            // Populate temp array of system constants for all possible VFDs
	            #arrIoDeviceIds[1] := "RackPumpVFD_1~PROFINET_interface~IODevice";
	            #arrIoDeviceIds[2] := "RackPumpVFD_2~PROFINET_interface~IODevice";
	            #arrIoDeviceIds[3] := "RackPumpVFD_3~PROFINET_interface~IODevice";
	            #arrIoDeviceIds[4] := "RackPumpVFD_4~PROFINET_interface~IODevice";
	            #arrIoDeviceIds[5] := "RackPumpVFD_5~PROFINET_interface~IODevice";
	            #arrIoDeviceIds[6] := "RackPumpVFD_6~PROFINET_interface~IODevice";
	            (*
	            #arrIoDeviceIds[7] := "RackPumpVFD_7~PROFINET_interface~IODevice";
	            #arrIoDeviceIds[8] := "RackPumpVFD_8~PROFINET_interface~IODevice";
	            #arrIoDeviceIds[9] := "RackPumpVFD_9~PROFINET_interface~IODevice";
	            #arrIoDeviceIds[10] := "RackPumpVFD_10~PROFINET_interface~IODevice";
	            #arrIoDeviceIds[11] := "RackPumpVFD_11~PROFINET_interface~IODevice";
	            #arrIoDeviceIds[12] := "RackPumpVFD_12~PROFINET_interface~IODevice";
	            
	            
	            #arrIoDeviceIds[13] := "RackPumpVFD_13~PROFINET_interface~IODevice";
	            #arrIoDeviceIds[14] := "RackPumpVFD_14~PROFINET_interface~IODevice";
	            #arrIoDeviceIds[15] := "RackPumpVFD_15~PROFINET_interface~IODevice";
	            #arrIoDeviceIds[16] := "RackPumpVFD_16~PROFINET_interface~IODevice";
	            #arrIoDeviceIds[17] := "RackPumpVFD_17~PROFINET_interface~IODevice";
	            #arrIoDeviceIds[18] := "RackPumpVFD_18~PROFINET_interface~IODevice";
	            #arrIoDeviceIds[19] := "RackPumpVFD_19~PROFINET_interface~IODevice";
	            #arrIoDeviceIds[20] := "RackPumpVFD_20~PROFINET_interface~IODevice";
	            #arrIoDeviceIds[21] := "RackPumpVFD_21~PROFINET_interface~IODevice";
	            #arrIoDeviceIds[22] := "RackPumpVFD_22~PROFINET_interface~IODevice";
	            #arrIoDeviceIds[23] := "RackPumpVFD_23~PROFINET_interface~IODevice";
	            #arrIoDeviceIds[24] := "RackPumpVFD_24~PROFINET_interface~IODevice";
	            #arrIoDeviceIds[25] := "RackPumpVFD_25~PROFINET_interface~IODevice";
	            #arrIoDeviceIds[26] := "RackPumpVFD_26~PROFINET_interface~IODevice";
	            #arrIoDeviceIds[27] := "RackPumpVFD_27~PROFINET_interface~IODevice";
	            #arrIoDeviceIds[28] := "RackPumpVFD_28~PROFINET_interface~IODevice";
	            #arrIoDeviceIds[29] := "RackPumpVFD_29~PROFINET_interface~IODevice";
	            #arrIoDeviceIds[30] := "RackPumpVFD_30~PROFINET_interface~IODevice";
	            *)
	            
	        END_REGION
	        
	        REGION Map VFD telegram hw submodule system constants
	            // Populate temp array of system constants for all possible VFDs
	            #arrTelegrams[1] := "RackPumpVFD_1~PROFINET_interface~Free_telegram";
	            #arrTelegrams[2] := "RackPumpVFD_2~PROFINET_interface~Free_telegram";
	            #arrTelegrams[3] := "RackPumpVFD_3~PROFINET_interface~Free_telegram";
	            #arrTelegrams[4] := "RackPumpVFD_4~PROFINET_interface~Free_telegram";
	            #arrTelegrams[5] := "RackPumpVFD_5~PROFINET_interface~Free_telegram";
	            #arrTelegrams[6] := "RackPumpVFD_6~PROFINET_interface~Free_telegram";
	            (*
	            #arrTelegrams[7] := "RackPumpVFD_7~PROFINET_interface~Free_telegram";
	            #arrTelegrams[8] := "RackPumpVFD_8~PROFINET_interface~Free_telegram";
	            #arrTelegrams[9] := "RackPumpVFD_9~PROFINET_interface~Free_telegram";
	            #arrTelegrams[10] := "RackPumpVFD_10~PROFINET_interface~Free_telegram";
	            #arrTelegrams[11] := "RackPumpVFD_11~PROFINET_interface~Free_telegram";
	            #arrTelegrams[12] := "RackPumpVFD_12~PROFINET_interface~Free_telegram";
	            
	            
	            #arrTelegrams[13] := "RackPumpVFD_13~PROFINET_interface~Free_telegram";
	            #arrTelegrams[14] := "RackPumpVFD_14~PROFINET_interface~Free_telegram";
	            #arrTelegrams[15] := "RackPumpVFD_15~PROFINET_interface~Free_telegram";
	            #arrTelegrams[16] := "RackPumpVFD_16~PROFINET_interface~Free_telegram";
	            #arrTelegrams[17] := "RackPumpVFD_17~PROFINET_interface~Free_telegram";
	            #arrTelegrams[18] := "RackPumpVFD_18~PROFINET_interface~Free_telegram";
	            #arrTelegrams[19] := "RackPumpVFD_19~PROFINET_interface~Free_telegram";
	            #arrTelegrams[20] := "RackPumpVFD_20~PROFINET_interface~Free_telegram";
	            #arrTelegrams[21] := "RackPumpVFD_21~PROFINET_interface~Free_telegram";
	            #arrTelegrams[22] := "RackPumpVFD_22~PROFINET_interface~Free_telegram";
	            #arrTelegrams[23] := "RackPumpVFD_23~PROFINET_interface~Free_telegram";
	            #arrTelegrams[24] := "RackPumpVFD_24~PROFINET_interface~Free_telegram";
	            #arrTelegrams[25] := "RackPumpVFD_25~PROFINET_interface~Free_telegram";
	            #arrTelegrams[26] := "RackPumpVFD_26~PROFINET_interface~Free_telegram";
	            #arrTelegrams[27] := "RackPumpVFD_27~PROFINET_interface~Free_telegram";
	            #arrTelegrams[28] := "RackPumpVFD_28~PROFINET_interface~Free_telegram";
	            #arrTelegrams[29] := "RackPumpVFD_29~PROFINET_interface~Free_telegram";
	            #arrTelegrams[30] := "RackPumpVFD_30~PROFINET_interface~Free_telegram";
	            *)
	            
	        END_REGION
	        
	        REGION Assign VFDs to racks, set up IO reconfig array
	            
	            #iVfdCount := 0;
	            
	            FOR #iRoomIndex := 1 TO #iNumRooms DO
	                
	                // Assign VFDs to configured rooms and racks, only using the ones we need
	                // Link up the Hw_SubModule system constant for each VFD's Profinet telegram
	                
	                FOR #iRackIndex := 1 TO #Controls.arrSetNumRacksPerRoom[#iRoomIndex] DO
	                    #iVfdCount += 1;
	                    
	                    "dbMain".Room[#iRoomIndex].Rack[#iRackIndex].Fertigation.Pump.fbVFD.hwInTelegram :=
	                    #arrTelegrams[#iVfdCount];
	                    
	                END_FOR;
	                
	            END_FOR;
	            
	            // populate data record array for reconfig io fb
	            #arrVfdDeviceConfig[-2] := 16#0100; // Version of the data record (1.0)
	            #arrVfdDeviceConfig[-1] := INT_TO_WORD(#iVfdCount); // Number of IO devices to be activated
	            
	            // populate input array with IO device IDs for all the VFDs we are using
	            FOR #i := 0 TO #iVfdCount-1 DO
	                #arrVfdDeviceConfig[#i] := UINT_TO_WORD(#arrIoDeviceIds[#i+1]);
	            END_FOR;
	            
	            // zero out rest of array (zero port interconnections used since everything is defined in topology)
	            FOR #i := #iVfdCount TO UINT_TO_INT("MAX_VFDS") DO
	                #arrVfdDeviceConfig[#i] := 0;
	            END_FOR;
	            
	        END_REGION
	        
	        REGION Assign Modbus TCP HVAC servers to rooms
	            FOR #i := 1 TO #iNumRooms DO
	                
	                // Port and connection ID
	                "dbMain".Room[#i].HVAC.Config.ID := INT_TO_UINT(80 + #i);
	                
	                // IP address
	                "dbMain".Room[#i].HVAC.Config.ModbusServerAddr.ADDR[1] := 10;
	                "dbMain".Room[#i].HVAC.Config.ModbusServerAddr.ADDR[2] := 1;
	                "dbMain".Room[#i].HVAC.Config.ModbusServerAddr.ADDR[3] := 0;
	                "dbMain".Room[#i].HVAC.Config.ModbusServerAddr.ADDR[4] := INT_TO_BYTE(19 + #i);
	                
	            END_FOR;
	        END_REGION
	        
	        IF #bInSimulation THEN
	            #iNextStep := #eStep_Done;
	        ELSE
	            #iNextStep := #eStep_Deactivate;
	        END_IF;
	        
	    END_IF;
	END_REGION
	
	REGION Call ReconfigIOSystem FB
	
	    CASE #iStep OF
	        #eStep_Deactivate:
	            #ReconfigIOSystem.REQ := TRUE;
	            #ReconfigIOSystem.MODE := 1;
	            IF #ReconfigIOSystem.DONE THEN
	                #iNextStep := #eStep_WaitForDeactivate;
	            END_IF;
	            
	        #eStep_WaitForDeactivate:
	            #ReconfigIOSystem.REQ := FALSE;
	            #iNextStep := #eStep_Reconfig;
	            
	        #eStep_Reconfig:
	            #ReconfigIOSystem.REQ := TRUE;
	            #ReconfigIOSystem.MODE := 2;
	            IF #ReconfigIOSystem.DONE THEN
	                #iNextStep := #eStep_WaitForReconfig;
	            END_IF;
	            
	        #eStep_WaitForReconfig:
	            #ReconfigIOSystem.REQ := FALSE;
	            #iNextStep := #eStep_Restart;
	            
	        #eStep_Restart:
	            #ReconfigIOSystem.REQ := TRUE;
	            #ReconfigIOSystem.MODE := 3;
	            IF #ReconfigIOSystem.DONE THEN
	                #iNextStep := #eStep_Done;
	            END_IF;
	                
	        ELSE
	            #ReconfigIOSystem.REQ := FALSE;
	            #ReconfigIOSystem.MODE := 0;
	            
	    END_CASE;
	    
	    #ReconfigIOSystem(REQ := #ReconfigIOSystem.REQ,
	                      MODE := #ReconfigIOSystem.MODE,
	                      LADDR := "Local~PROFINET_interface_1",
	                      CTRLREC := #arrVfdDeviceConfig,
	                      STATUS => #ReconfigIOSystem.STATUS,
	                      BUSY => #ReconfigIOSystem.BUSY,
	                      DONE => #ReconfigIOSystem.DONE,
	                      ERROR => #ReconfigIOSystem.ERROR);
	    
	    // catch and log error
	    IF #ReconfigIOSystem.ERROR THEN
	        #Status.ErrorMsg := CONCAT(IN1 := #Status.ErrorMsg, IN2 := ' ReconfigIO Error Code: ');
	        #retVal := HTA(IN := #ReconfigIOSystem.STATUS, N := 4, OUT => #strErrorCode);
	        #Status.ErrorMsg := CONCAT(IN1 := #Status.ErrorMsg, IN2 := #strErrorCode);
	        
	        #Status.ErrorMsg := CONCAT(IN1 := #Status.ErrorMsg, IN2 := ' On device: ');
	        #retVal := HTA(IN := #ReconfigIOSystem.ERR_INFO, N := 2, OUT => #strErrorCode);
	        #Status.ErrorMsg := CONCAT(IN1 := #Status.ErrorMsg, IN2 := #strErrorCode);
	        
	        #iNextStep := #eStep_Error;
	    END_IF;
	    
	END_REGION
	
	REGION Set status outputs
	    #Status.bDone := #iStep = #eStep_Done;
	    #Status.bBusy := #iStep <> #eStep_Done AND #iStep <> #eStep_Error;
	    #Status.bError := #iStep = #eStep_Error;
	    
	END_REGION
	
	// set step for next scan
	#iStep := #iNextStep;
END_FUNCTION_BLOCK

FUNCTION_BLOCK "fbRoom"   // FB3, LAD
{ S7_Optimized_Access := 'TRUE' }
VERSION : 0.1
// stored: AutoNumber true, IsIECCheckEnabled false, IsRetainMemResEnabled false, MemoryReserve 100, SetENOAutomatically false, UDAEnableTagReadback false
   VAR_INPUT
      arrAI { ExternalAccessible := 'False'; ExternalVisible := 'False'; ExternalWritable := 'False'} : Array[1.."NUM_AI_ROOM"] of Int;
      AI AT arrAI : "udtRoomAI";
   END_VAR
   VAR_OUTPUT
      arrDQ { ExternalAccessible := 'False'; ExternalVisible := 'False'; ExternalWritable := 'False'} : Array[1.."NUM_DQ_ROOM"] of Bool;
      DQ AT arrDQ : "udtRoomDQ";
   END_VAR
   VAR
      Rack { ExternalVisible := 'False'} : Array[1.."MAX_RACKS_PER_ROOM"] of "fbRack";
      Fertigation { ExternalVisible := 'False'} : "fbRoomFertigation";
      HVAC { ExternalVisible := 'False'} : "fbRoomHVAC";
   END_VAR
   VAR RETAIN
      Config { ExternalVisible := 'False'; ExternalWritable := 'False'} : Struct
         iNumRacks { ExternalVisible := 'False'; ExternalWritable := 'False'} : Int := 1;
      END_STRUCT;
   END_VAR
   VAR
      AI_Temperature_1 { ExternalVisible := 'False'} : "fbAlarmedSetpoint";
      AI_Temperature_2 { ExternalVisible := 'False'} : "fbAlarmedSetpoint";
      AI_Humidity_1 { ExternalVisible := 'False'} : "fbAlarmedSetpoint";
      AI_Humidity_2 { ExternalVisible := 'False'} : "fbAlarmedSetpoint";
      AI_TankLevel { ExternalVisible := 'False'} : "fbAlarmedSetpoint";
      AI_NutrientALevel { ExternalVisible := 'False'} : "fbAlarmedSetpoint";
      AI_NutrientBLevel { ExternalVisible := 'False'} : "fbAlarmedSetpoint";
      AI_NutrientAcidLevel { ExternalVisible := 'False'} : "fbAlarmedSetpoint";
      AI_pHSensor { ExternalVisible := 'False'} : "fbAlarmedSetpoint";
      AI_ECSensor { ExternalVisible := 'False'} : "fbAlarmedSetpoint";
      AI_ISESensor { ExternalVisible := 'False'} : "fbAlarmedSetpoint";
      AI_ORPSensor { ExternalVisible := 'False'} : "fbAlarmedSetpoint";
   END_VAR
   VAR RETAIN
      DQ_MPathSolenoid { ExternalVisible := 'False'} : "udtDigitalOutput";
      DQ_FreshWaterSolenoid { ExternalVisible := 'False'} : "udtDigitalOutput";
      DQ_DischargeSolenoid { ExternalVisible := 'False'} : "udtDigitalOutput";
      DQ_TankReturnSolenoid { ExternalVisible := 'False'} : "udtDigitalOutput";
      DQ_NutrientA { ExternalVisible := 'False'} : "udtDigitalOutput";
      DQ_NutrientB { ExternalVisible := 'False'} : "udtDigitalOutput";
      DQ_NutrientAcid { ExternalVisible := 'False'} : "udtDigitalOutput";
      DQ_NutrientMixing { ExternalVisible := 'False'} : "udtDigitalOutput";
      DQ_CO2Solenoid { ExternalVisible := 'False'} : "udtDigitalOutput";
   END_VAR
   VAR
      arrFertigationSettings { ExternalAccessible := 'False'; ExternalVisible := 'False'; ExternalWritable := 'False'} : Array[0.."MAX_RACKS_PER_ROOM"] of "udtFertigationSettings";
   END_VAR
   VAR_TEMP
      i : Int;   // Index for iterating through racks
      max_temp : Int;
   END_VAR
   // AI_Temperature_1.Config.rLowCalibration := -40.0;
   // AI_Temperature_1.Config.rHighCalibration := 140.0;
   // AI_Temperature_2.Config.rLowCalibration := -40.0;
   // AI_Temperature_2.Config.rHighCalibration := 140.0;
   // AI_Humidity_1.Config.rLowCalibration := 0.0;
   // AI_Humidity_1.Config.rHighCalibration := 100.0;
   // AI_Humidity_2.Config.rLowCalibration := 0.0;
   // AI_Humidity_2.Config.rHighCalibration := 100.0;
   // AI_TankLevel.Config.rLowCalibration := 0.0;
   // AI_TankLevel.Config.rHighCalibration := 1085.0;
   // AI_NutrientALevel.Config.rLowCalibration := 0.0;
   // AI_NutrientALevel.Config.rHighCalibration := 200.0;
   // AI_NutrientBLevel.Config.rLowCalibration := 0.0;
   // AI_NutrientBLevel.Config.rHighCalibration := 200.0;
   // AI_NutrientAcidLevel.Config.rLowCalibration := 0.0;
   // AI_NutrientAcidLevel.Config.rHighCalibration := 200.0;
   // AI_pHSensor.Config.rLowCalibration := 0.0;
   // AI_pHSensor.Config.rHighCalibration := 14.0;
   // AI_ECSensor.Config.rLowCalibration := 0.0;
   // AI_ECSensor.Config.rHighCalibration := 5.0;
   // AI_ISESensor.Config.rLowCalibration := 0.0;
   // AI_ISESensor.Config.rHighCalibration := 10000.0;
   // AI_ORPSensor.Config.rLowCalibration := -1500.0;
   // AI_ORPSensor.Config.rHighCalibration := 1500.0;
BEGIN

REGION Network 1 (SCL): Process room-level analog inputs
   #AI_Temperature_1(#AI.IW_RoomTemperature_1);
   #AI_Temperature_2(#AI.IW_RoomTemperature_2);
   #AI_Humidity_1(#AI.IW_RoomHumidity_1);
   #AI_Humidity_2(#AI.IW_RoomHumidity_2);
   #AI_TankLevel(#AI.IW_TankLevel);
   #AI_NutrientALevel(#AI.IW_NutrientALevel);
   #AI_NutrientBLevel(#AI.IW_NutrientBLevel);
   #AI_NutrientAcidLevel(#AI.IW_NutrientAcidLevel);
   #AI_pHSensor(#AI.IW_pHSensor);
   #AI_ECSensor(#AI.IW_ECSensor);
   #AI_ISESensor(#AI.IW_ISESensor);
   #AI_ORPSensor(#AI.IW_ORPSensor);
   //#AI_CO2Sensor(#AI.IW_CO2Sensor);
END_REGION

REGION Network 2 (SCL): Call rack FBs
   #max_temp := MAX(IN1 := #AI_Temperature_1.rActual, IN2 := #AI_Temperature_2.rActual);
   #max_temp := MAX(IN1 := #max_temp, IN2 := #HVAC.Temperature_Cooling.rActual);

   FOR #i := 1 TO #Config.iNumRacks DO

       #Rack[#i](iInMutexLockConfirmation := #Fertigation.arrOutMutexLocks[#i],
                 udtInLastNutrientReading := #Fertigation.arrOutNutrientReading[#i],
                 bInSupplySolenoidFromRoomFertigation := #Fertigation.arrOutSupplySolenoids[#i],
                 bInReturnSolenoidFromRoomFertigation := #Fertigation.arrOutReturnSolenoids[#i],
                 iInLightsDelaySecs := #i * 5000, // delay each rack by 5 seconds to prevent current spike
                 arrAI := #Rack[#i].arrAI,
                 rInCurrentTemperature := #max_temp,
                 iOutMutexRequest => #Fertigation.arrInMutexRequests[#i],
                 OutFertigationSettings => #arrFertigationSettings[#i],
                 arrDQ => #Rack[#i].arrDQ);
   END_FOR;
END_REGION

REGION Network 3 (SCL): Call room-level fertigation control logic and map rack supply and return solenoids
   #Fertigation(arrInMutexRequests:=#Fertigation.arrInMutexRequests,
                arrInFertigationSettings:=#arrFertigationSettings,
                rInTankLevel:=#AI_TankLevel.rActual,
                rInNutrientALevel:=#AI_NutrientALevel.rActual,
                rInNutrientBLevel:=#AI_NutrientBLevel.rActual,
                rInNutrientAcidLevel:=#AI_NutrientAcidLevel.rActual,
                rInpHSensor:=#AI_pHSensor.rActual,
                rInECSensor:=#AI_ECSensor.rActual,
                rInISESensor:=#AI_ISESensor.rActual,
                rInORPReading:=#AI_ORPSensor.rActual,
                iInNumRacks:=#Config.iNumRacks,
                bOutTankReturnSolenoid=>#Fertigation.bOutTankReturnSolenoid,
                bOutMPathSolenoid=>#Fertigation.bOutMPathSolenoid,
                bOutFreshWaterSolenoid=>#Fertigation.bOutFreshWaterSolenoid,
                bOutDischargeSolenoid=>#Fertigation.bOutDischargeSolenoid,
                bOutNutrientMixing=>#Fertigation.bOutNutrientMixing,
                bOutNutrientA=>#Fertigation.bOutNutrientA,
                bOutNutrientB=>#Fertigation.bOutNutrientB,
                bOutNutrientAcid=>#Fertigation.bOutNutrientAcid,
                arrOutNutrientReading=>#Fertigation.arrOutNutrientReading,
                arrOutMutexLocks=>#Fertigation.arrOutMutexLocks,
                arrOutSupplySolenoids=>#Fertigation.arrOutSupplySolenoids,
                arrOutReturnSolenoids=>#Fertigation.arrOutReturnSolenoids);
END_REGION

REGION Network 4 (SCL): Call HVAC and CO2 control logic
   #HVAC(iInCO2ReadingRaw := #AI.IW_CO2Sensor,
         bOutCO2Solenoid=>#HVAC.bOutCO2Solenoid);
END_REGION

REGION Network 5 (SCL): Set room-level outputs
   #DQ.Q_MPathSolenoid := "fcDigitalOutput"(bInAutoVal := #Fertigation.bOutMPathSolenoid, InOutUdt := #DQ_MPathSolenoid);
   #DQ.Q_FreshWaterSolenoid := "fcDigitalOutput"(bInAutoVal := #Fertigation.bOutFreshWaterSolenoid, InOutUdt := #DQ_FreshWaterSolenoid);
   #DQ.Q_DischargeSolenoid := "fcDigitalOutput"(bInAutoVal := #Fertigation.bOutDischargeSolenoid, InOutUdt := #DQ_DischargeSolenoid);
   #DQ.Q_TankReturnSolenoid := "fcDigitalOutput"(bInAutoVal := #Fertigation.bOutTankReturnSolenoid, InOutUdt := #DQ_TankReturnSolenoid);
   #DQ.Q_NutrientAEnable := "fcDigitalOutput"(bInAutoVal := #Fertigation.bOutNutrientA, InOutUdt := #DQ_NutrientA);
   #DQ.Q_NutrientBEnable := "fcDigitalOutput"(bInAutoVal := #Fertigation.bOutNutrientB, InOutUdt := #DQ_NutrientB);
   #DQ.Q_NutrientAcidEnable := "fcDigitalOutput"(bInAutoVal := #Fertigation.bOutNutrientAcid, InOutUdt := #DQ_NutrientAcid);
   #DQ.Q_NutrientMixingPumps := "fcDigitalOutput"(bInAutoVal := #Fertigation.bOutNutrientMixing, InOutUdt := #DQ_NutrientMixing);

   #DQ.Q_CO2Solenoid := "fcDigitalOutput"(bInAutoVal := #HVAC.bOutCO2Solenoid, InOutUdt := #DQ_CO2Solenoid);
END_REGION
END_FUNCTION_BLOCK

FUNCTION_BLOCK "fbAlarmedSetpoint"   // FB1, LAD
{ S7_Optimized_Access := 'TRUE' }
VERSION : 0.1
// Processes raw analog input and evaluates alarms.
// Note: All alarms are momentary, i.e. no ack necessary and they reset themselves when the condition becomes false.
// stored: AutoNumber true, IsIECCheckEnabled false, IsRetainMemResEnabled false, MemoryReserve 100, SetENOAutomatically false, UDAEnableTagReadback false
   VAR_INPUT
      iInRawValue { ExternalAccessible := 'False'; ExternalVisible := 'False'; ExternalWritable := 'False'} : Int;
   END_VAR
   VAR RETAIN
      arrSetpoints { ExternalVisible := 'False'} : Array[1..10] of "udtTimeOfDaySetpoint";   // Setpoints need to be chronologically increasing
      rSetpoint { ExternalVisible := 'False'; ExternalWritable := 'False'} : Real;
      rActual { ExternalVisible := 'False'; ExternalWritable := 'False'} : Real;
      Alarms { ExternalVisible := 'False'; ExternalWritable := 'False'} : Struct
         bHigh { ExternalVisible := 'False'; ExternalWritable := 'False'} : Bool;   // rActual exceeds limit
         bLow { ExternalVisible := 'False'; ExternalWritable := 'False'} : Bool;   // rActual exceeds limit
         bRate { ExternalVisible := 'False'; ExternalWritable := 'False'} : Bool;   // rActual increases or decreases faster than the limit. False if rate is left as 0.
         bSetpoint { ExternalVisible := 'False'; ExternalWritable := 'False'} : Bool;   // rActual does not reach rSetpoint within allowed time delay and deadband. False if deadband left at 0.
      END_STRUCT;
      Config { ExternalVisible := 'False'} : Struct
         rLowCalibration { ExternalVisible := 'False'} : Real := 0.0;
         rHighCalibration { ExternalVisible := 'False'} : Real := 100.0;
         Alarms { ExternalVisible := 'False'} : Struct
            rLowLimit { ExternalVisible := 'False'} : Real := 0.0;
            rHighLimit { ExternalVisible := 'False'} : Real := 100.0;
            rRateLimit { ExternalVisible := 'False'} : Real;   // Maximum permitted change in rActual per second
            rDeadband { ExternalVisible := 'False'} : Real;   // Range around rSetpoint that is still considered within range
            iSettlingSecs { ExternalVisible := 'False'} : Int;   // Allowable delay to allow rActual to reach rSetpoint after change
         END_STRUCT;
      END_STRUCT;
   END_VAR
   VAR
      TON_RateCheck { ExternalAccessible := 'False'; ExternalVisible := 'False'; ExternalWritable := 'False'} : TON_TIME;
      rActual_Prev { ExternalAccessible := 'False'; ExternalVisible := 'False'; ExternalWritable := 'False'} : Real;
      TON_Settling { ExternalAccessible := 'False'; ExternalVisible := 'False'; ExternalWritable := 'False'} : TON_TIME;
      rSetpoint_Prev { ExternalAccessible := 'False'; ExternalVisible := 'False'; ExternalWritable := 'False'} : Real;
   END_VAR
   VAR_TEMP
      localTime : Date_And_Time;
      ret_val : Int;
      currentTOD : Time_Of_Day;
      i : Int;
      currentTODsecs : DInt;
   END_VAR
   VAR_TEMP   // added for the SCL form of the ladder/FBD networks
      _w1 : Bool;
      _w2 : Bool;
   END_VAR
BEGIN

REGION Network 1 (SCL): Scale raw input based on calibration
   #rActual := "fcAnalogInput"(iInRawValue := #iInRawValue,
                               rLowCalibration := #Config.rLowCalibration,
                               rHighCalibration := #Config.rHighCalibration);
END_REGION

REGION Network 2 (SCL): Low/high alarms
   #Alarms.bHigh := #rActual > #Config.Alarms.rHighLimit;
   #Alarms.bLow  := #rActual < #Config.Alarms.rLowLimit;
END_REGION

REGION Network 3 (SCL): Rate of change alarm
   // Set the current value on startup to prevent a spurious alarm
   IF "FirstScan" THEN
       #rActual_Prev := #rActual;
   END_IF;

   // Compare values at every given time interval to get rate of change
   IF #TON_RateCheck.Q THEN
       #Alarms.bRate := ( ABS(#rActual - #rActual_Prev) > #Config.Alarms.rRateLimit)
       AND (#Config.Alarms.rRateLimit <> 0.0); // ignore alarm if max rate is left at default of 0

       #rActual_Prev := #rActual;
   END_IF;

   #TON_RateCheck(IN := NOT #TON_RateCheck.Q,
                  PT := t#1s);
END_REGION

REGION Network 4: Get current time of day
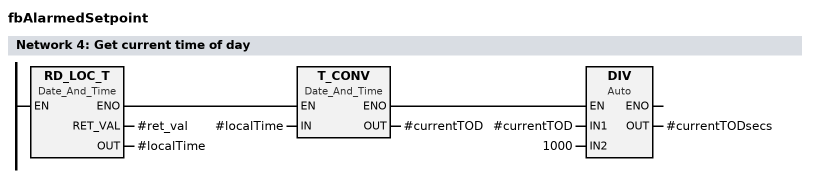
   RUNG wire#powerrail
      { S7_Templates := "date_type := Date_And_Time" } RD_LOC_T(RET_VAL => #ret_val, OUT => #localTime)
      { S7_Templates := "[src_type := Date_And_Time, dest_type := Time_Of_Day]" } T_CONV(IN := #localTime, OUT => #currentTOD)
      Div(in1 := #currentTOD, in2 := 1000, out => #currentTODsecs)
   END_RUNG
   // the same network as SCL:
   #ret_val := RD_LOC_T(OUT => #localTime, ENO => #_w1);
   T_CONV(EN := #_w1, IN := #localTime, OUT => #currentTOD, ENO => #_w2);
   IF #_w2 THEN #currentTODsecs := #currentTOD / 1000; END_IF;
END_REGION

REGION Network 5 (SCL): Determine current setpoint based on time of day
   IF #arrSetpoints[1].TimeOfDaySeconds = -1 THEN
       // If no time schedule is defined, default to first setpoint in array
       #rSetpoint := #arrSetpoints[1].rSetpoint;

   ELSIF #currentTODsecs < #arrSetpoints[1].TimeOfDaySeconds THEN
       // Check for setpoint from previous day
       FOR #i := 10 TO 1 BY -1 DO
           IF #arrSetpoints[#i].TimeOfDaySeconds <> -1 THEN
               #rSetpoint := #arrSetpoints[#i].rSetpoint;
               EXIT;
           END_IF;
       END_FOR;

   ELSE
       // Iterate through and find current setpoint
       FOR #i := 1 TO 9 DO
           IF #currentTODsecs < #arrSetpoints[#i + 1].TimeOfDaySeconds OR #arrSetpoints[#i + 1].TimeOfDaySeconds = -1 THEN
               #rSetpoint := #arrSetpoints[#i].rSetpoint;
               EXIT;
           ELSIF #i = 9 THEN
               #rSetpoint := #arrSetpoints[10].rSetpoint;
           END_IF;
       END_FOR;

   END_IF;
END_REGION

REGION Network 6 (SCL): Setpoint not reached alarm


   // Set the current value on startup to prevent a spurious alarm
   IF "FirstScan" THEN
       #rSetpoint_Prev := #rSetpoint;
   END_IF;

   // Evaluate alarm after settling time has elapsed
   #TON_Settling(IN := (#rSetpoint = #rSetpoint_Prev), // restart timer when setpoint changes
                 PT := INT_TO_TIME(#Config.Alarms.iSettlingSecs * 1000)); // convert to ms

   #Alarms.bSetpoint := #TON_Settling.Q AND (
   (#rActual < #rSetpoint - #Config.Alarms.rDeadband / 2.0) OR
   (#rActual > #rSetpoint + #Config.Alarms.rDeadband / 2.0) )
   AND (#Config.Alarms.rDeadband <> 0.0); // ignore alarm if deadband is left at default of 0

   // Save setpoint value for next comparison
   #rSetpoint_Prev := #rSetpoint;
END_REGION
END_FUNCTION_BLOCK

FUNCTION_BLOCK "fbRack"   // FB5, LAD
{ S7_Optimized_Access := 'TRUE' }
VERSION : 0.1
// stored: AutoNumber true, IsIECCheckEnabled false, IsRetainMemResEnabled false, MemoryReserve 100, SetENOAutomatically false, UDAEnableTagReadback false
   VAR_INPUT
      iInMutexLockConfirmation { ExternalAccessible := 'False'; ExternalVisible := 'False'; ExternalWritable := 'False'} : Int;
      udtInLastNutrientReading { ExternalAccessible := 'False'; ExternalVisible := 'False'; ExternalWritable := 'False'} : "udtNutrientReading";
      bInSupplySolenoidFromRoomFertigation { ExternalAccessible := 'False'; ExternalVisible := 'False'; ExternalWritable := 'False'} : Bool;
      bInReturnSolenoidFromRoomFertigation { ExternalAccessible := 'False'; ExternalVisible := 'False'; ExternalWritable := 'False'} : Bool;
      iInLightsDelaySecs { ExternalAccessible := 'False'; ExternalVisible := 'False'; ExternalWritable := 'False'} : Int;
      rInCurrentTemperature : Real;
      arrAI { ExternalAccessible := 'False'; ExternalVisible := 'False'; ExternalWritable := 'False'} : Array[1.."NUM_AI_RACK"] of Int;
      AI AT arrAI : "udtRackAI";
   END_VAR
   VAR_OUTPUT
      iOutMutexRequest { ExternalAccessible := 'False'; ExternalVisible := 'False'; ExternalWritable := 'False'} : Int;
      OutFertigationSettings { ExternalAccessible := 'False'; ExternalVisible := 'False'; ExternalWritable := 'False'} : "udtFertigationSettings";
      arrDQ { ExternalAccessible := 'False'; ExternalVisible := 'False'; ExternalWritable := 'False'} : Array[1.."NUM_DQ_RACK"] of Bool;
      DQ AT arrDQ : "udtRackDQ";
   END_VAR
   VAR
      Lighting { ExternalVisible := 'False'} : "fbRackLights";
      Fertigation { ExternalVisible := 'False'} : "fbRackFertigation";
      AI_ReservoirLevel { ExternalVisible := 'False'} : "fbAlarmedSetpoint";
   END_VAR
   VAR RETAIN
      DQ_SupplySolenoid { ExternalVisible := 'False'} : "udtDigitalOutput";
      DQ_ReturnSolenoid { ExternalVisible := 'False'} : "udtDigitalOutput";
      DQ_ShelfSolenoid { ExternalVisible := 'False'} : "udtDigitalOutput";
      DQ_Lights { ExternalVisible := 'False'} : "udtDigitalOutput";
   END_VAR
   // AI_ReservoirLevel.Config.rLowCalibration := 0.0;
   // AI_ReservoirLevel.Config.rHighCalibration := 951.0;
BEGIN

REGION Network 1 (SCL)
   // Note that rack supply/return solenoids are managed by room-level fertigation FB
   // Process rack-level analog inputs
   #AI_ReservoirLevel(#AI.IW_ReservoirLevel);

   // Call lighting control fb
   #Lighting(iInDelaySecs := #iInLightsDelaySecs,
             rInCurrentTemperature := #rInCurrentTemperature,
             bOutLights => #Lighting.bOutLights);

   // Call rack-level fertigation logic
   #Fertigation(iInMutexLockConfirmation := #iInMutexLockConfirmation,
                InLastNutrientReading:= #udtInLastNutrientReading,
                rInReservoirLevel := #AI_ReservoirLevel.rActual,
                bInReturnSolenoidStatus:=#DQ.Q_ReturnSolenoid,
                bInShelfSolenoidStatus:=#DQ.Q_ShelfSolenoid,
                iOutMutexRequest => #iOutMutexRequest,
                OutFertigationSettings => #OutFertigationSettings,
                bOutShelfSolenoid => #Fertigation.bOutShelfSolenoid);

   // Set rack-level outputs
   // Rack supply/return solenoids are managed by room-level fertigation FB
   #DQ.Q_SupplySolenoid := "fcDigitalOutput"(bInAutoVal := #bInSupplySolenoidFromRoomFertigation, InOutUdt := #DQ_SupplySolenoid);
   #DQ.Q_ReturnSolenoid := "fcDigitalOutput"(bInAutoVal := #bInReturnSolenoidFromRoomFertigation, InOutUdt := #DQ_ReturnSolenoid);
   #DQ.Q_ShelfSolenoid  := "fcDigitalOutput"(bInAutoVal := #Fertigation.bOutShelfSolenoid, InOutUdt := #DQ_ShelfSolenoid);
   #DQ.Q_Lights         := "fcDigitalOutput"(bInAutoVal := #Lighting.bOutLights, InOutUdt := #DQ_Lights);
END_REGION
END_FUNCTION_BLOCK

FUNCTION_BLOCK "fbRackLights"   // FB6, LAD
{ S7_Optimized_Access := 'TRUE' }
VERSION : 0.1
// stored: AutoNumber true, IsIECCheckEnabled false, IsRetainMemResEnabled false, MemoryReserve 100, SetENOAutomatically false, UDAEnableTagReadback false
   VAR_INPUT
      iInDelaySecs { ExternalAccessible := 'False'; ExternalVisible := 'False'; ExternalWritable := 'False'} : Int;
      rInCurrentTemperature : Real;
   END_VAR
   VAR_OUTPUT
      bOutLights { ExternalAccessible := 'False'; ExternalVisible := 'False'; ExternalWritable := 'False'} : Bool;
   END_VAR
   VAR RETAIN
      Controls { ExternalVisible := 'False'} : Struct
         iMode { ExternalVisible := 'False'} : Int;   // 0: Off, 1: On, 2: Auto
         diOffTime { ExternalVisible := 'False'} : DInt;   // Off time (seconds past midnight)
         diOnTime { ExternalVisible := 'False'} : DInt;   // On time (seconds past midnight)
         rHighTemperatureLimit { ExternalVisible := 'False'} : Real := 75.0;
      END_STRUCT;
      Status { ExternalVisible := 'False'; ExternalWritable := 'False'} : Struct
         diSecondsElapsed { ExternalVisible := 'False'; ExternalWritable := 'False'} : DInt;
      END_STRUCT;
   END_VAR
   VAR
      bLightsCommand { ExternalAccessible := 'False'; ExternalVisible := 'False'; ExternalWritable := 'False'} : Bool;
   END_VAR
   VAR RETAIN
      TON_OnDelay { ExternalAccessible := 'False'; ExternalVisible := 'False'; ExternalWritable := 'False'; S7_SetPoint := 'True'} : TON_TIME;
   END_VAR
   VAR_TEMP
      tCurrentDateTime : Date_And_Time;   // Current PLC Date and Time
      tCurrentTimeMilli : Time_Of_Day;   // Current time (ms since 0:00:00)
      retVal : Int;   // Garbage return value from RD_LOC_T
      diSeconds : DInt;
   END_VAR
   VAR CONSTANT
      eOffMode : Int := 0;
      eOnMode : Int := 1;
      eAutoMode : Int := 2;
   END_VAR
BEGIN

REGION Network 1 (SCL): State 0 - Off Mode and State 1 - On Mode
   // Directly assign rack light output based on off or on mode
   IF #Controls.iMode = #eOffMode THEN
       #bLightsCommand := 0;
   ELSIF #Controls.iMode = #eOnMode THEN
       #bLightsCommand := 1;
   END_IF;
END_REGION

REGION Network 2 (SCL): State 2 - Auto Mode
   // Check the current time against the on time and off time, and assign the lights appropriately
   IF #Controls.iMode = #eAutoMode THEN

       //Get current time from PLC and convert to seconds since 0:00:00
       #retVal := RD_LOC_T(OUT => #tCurrentDateTime);
       #tCurrentTimeMilli := DT_TO_TOD(IN := #tCurrentDateTime);
       #diSeconds := TOD_TO_DINT(IN := #tCurrentTimeMilli)/1000; //Go from ms time to DInt seconds

       // Situation 1: Off time happens after on time
       IF #Controls.diOffTime > #Controls.diOnTime THEN 
           IF #diSeconds > #Controls.diOnTime AND #diSeconds < #Controls.diOffTime THEN
               #bLightsCommand := 1;
           ELSE
               #bLightsCommand := 0;
           END_IF;

       // Situation 2: On time happens after off time
       ELSE
           IF #diSeconds > #Controls.diOffTime AND #diSeconds < #Controls.diOnTime THEN
               #bLightsCommand := 0;
           ELSE
               #bLightsCommand := 1;
           END_IF;
       END_IF;
   END_IF;
END_REGION

REGION Network 3 (SCL): Temperature Override When in Auto

   IF #Controls.iMode = #eAutoMode AND #rInCurrentTemperature > #Controls.rHighTemperatureLimit THEN
       #bLightsCommand := 0;
   END_IF;
END_REGION

REGION Network 4 (SCL): Write seconds elapsed status and set outputs with confugred delay
   #Status.diSecondsElapsed := #diSeconds;

   #TON_OnDelay(IN := #bLightsCommand,
                PT := INT_TO_TIME(#iInDelaySecs));

   #bOutLights := #TON_OnDelay.Q;
END_REGION
END_FUNCTION_BLOCK

FUNCTION_BLOCK "fbRackFertigation"
{ S7_Optimized_Access := 'TRUE' }
VERSION : 0.1
   VAR_INPUT 
      iInMutexLockConfirmation { ExternalAccessible := 'False'; ExternalVisible := 'False'; ExternalWritable := 'False'} : Int;   // 0: Off, 1: Fill, 2: Measurement/Dosing, 3:Discharge
      InLastNutrientReading { ExternalVisible := 'False'; ExternalWritable := 'False'} : "udtNutrientReading";
      rInReservoirLevel { ExternalAccessible := 'False'; ExternalVisible := 'False'; ExternalWritable := 'False'} : Real;   // Rack reservoir level
      bInReturnSolenoidStatus { ExternalAccessible := 'False'; ExternalVisible := 'False'; ExternalWritable := 'False'} : Bool;   // Return solenoid status for determining when return to main tank or discharge
      bInShelfSolenoidStatus { ExternalAccessible := 'False'; ExternalVisible := 'False'; ExternalWritable := 'False'} : Bool;
   END_VAR

   VAR_OUTPUT 
      iOutMutexRequest { ExternalAccessible := 'False'; ExternalVisible := 'False'; ExternalWritable := 'False'} : Int;   // 0: Off, 1: Fill, 2: Measurement/Dosing, 3:Discharge
      OutFertigationSettings { ExternalAccessible := 'False'; ExternalVisible := 'False'; ExternalWritable := 'False'} : "udtFertigationSettings";
      bOutShelfSolenoid { ExternalAccessible := 'False'; ExternalVisible := 'False'; ExternalWritable := 'False'} : Bool;
   END_VAR

   VAR RETAIN
      Controls { ExternalVisible := 'False'} : Struct
         iModeCommand { ExternalVisible := 'False'} : Int;   // 0: Off, 1: Fill, 2: Measurement/Dosing, 3:Discharge, 4: Circulate
         dtLastMeasurement { ExternalVisible := 'False'} : Date_And_Time := DT#2020-07-14-15:57:00;   // time since last measurement (0-86400s)
         bEndDischargeCommand { ExternalVisible := 'False'} : Bool;   // Command to end discharge before timer expires
         diDischargeTimeSecs { ExternalVisible := 'False'} : DInt := 10800;   // Discharge duration (seconds)
         rPumpReservoirInterlockLevel { ExternalVisible := 'False'} : Real := 180.0;   // Reservoir level below which to turn off pump (L)
         rPumpContinousSpeed { ExternalVisible := 'False'} : Real := 79.2;   // Commanded pump speed (%)
         rPumpReturnSpeed { ExternalVisible := 'False'} : Real := 80.8;   // Commanded pump speed (%)
         rPumpDischargeSpeed { ExternalVisible := 'False'} : Real := 91.7;   // Commanded pump speed (%)
         diMeasurementSecs { ExternalVisible := 'False'} : DInt := 180;   // Duration of measurement (seconds)
         diDosingIntervalMins { ExternalVisible := 'False'} : DInt := 120;   // Time to stay in circulate mode before trigerring a M&D routine
         rMeasurementVolume { ExternalVisible := 'False'} : Real := 200.0;   // Volume to move from reservoir to tank during measurement
         iISEModeCommand { ExternalVisible := 'False'} : Int := 1;   // 0: Off, 1: Load, 2: Deplete
         bNutrientAEnable { ExternalVisible := 'False'} : Bool := true;   // Enable nutrient A for dosing
         bNutrientBEnable { ExternalVisible := 'False'} : Bool := true;   // Enable nutrient B for dosing
         rISELowSP { ExternalVisible := 'False'} : Real := 35.0;   // Low ISE setpoint for dosing
         rISEHighSP { ExternalVisible := 'False'} : Real := 145.0;   // High ISE setpoint for dosing
         diNutrientDosingSecs { ExternalVisible := 'False'} : DInt := 60;   // Duration of nutrient dosing (seconds)
         rOperatingVolume { ExternalVisible := 'False'} : Real := 450.0;   // Operating volume for rack reservoir (L)
         rTotalShelfVolume { ExternalVisible := 'False'} : Real := 1800.0;   // Total volume of the shelves (L)
         rMaxReservoirVolume { ExternalVisible := 'False'} : Real := 900.0;   // Maximum water capacity of the rack reservoir (L)
      END_STRUCT;
      Status { ExternalVisible := 'False'; ExternalWritable := 'False'} : Struct
         iState { ExternalVisible := 'False'; ExternalWritable := 'False'} : Int;   // 0: Off, 1: Fill, 2: Measurement/Dosing, 3:Discharge, 4: Circulate
         NutrientLevels { ExternalVisible := 'False'; ExternalWritable := 'False'; S7_SetPoint := 'False'} : "udtNutrientReading";   // Last measured nutrient levels
      END_STRUCT;
   END_VAR
   VAR 
      Pump { ExternalVisible := 'False'; S7_SetPoint := 'False'} : "fbRackPump";
   END_VAR
   VAR RETAIN
      bShelfSolenoidCommand { ExternalAccessible := 'False'; ExternalVisible := 'False'; ExternalWritable := 'False'} : Bool;   // Command for shelf solenoid
      bLockConfirmedModeActive { ExternalAccessible := 'False'; ExternalVisible := 'False'; ExternalWritable := 'False'} : Bool;   // Memory bit for mutex lock, used to detect lock dropping out
      iNextMode { ExternalAccessible := 'False'; ExternalVisible := 'False'; ExternalWritable := 'False'} : Int;   // Holder for next user commanded mode
      rInitialVolume { ExternalAccessible := 'False'; ExternalVisible := 'False'; ExternalWritable := 'False'} : Real;   // Initial volume of reservoir at start of measurement
   END_VAR
   VAR 
      NutrientReadingReady {InstructionName := 'F_TRIG'; LibVersion := '1.0'; ExternalAccessible := 'False'; ExternalVisible := 'False'; ExternalWritable := 'False'; S7_SetPoint := 'False'} : F_TRIG;
   END_VAR
   VAR RETAIN
      TON_Circulate {InstructionName := 'TON_TIME'; LibVersion := '1.0'; ExternalAccessible := 'False'; ExternalVisible := 'False'; ExternalWritable := 'False'; S7_SetPoint := 'False'} : TON_TIME;
   END_VAR

   VAR_TEMP 
      retVal : Int;
      tCurrentDateTime : Date_And_Time;
      lastDelta : Date_And_Time;
      rPumpSpeed : Real;
   END_VAR

   VAR CONSTANT 
      eRackMode_Off : Int := 0;   // Rack Off State
      eRackMode_Fill : Int := 1;   // Rack Fill State
      eRackMode_MeasurementDosing : Int := 2;   // Rack Measurement and Dosing State
      eRackMode_Discharge : Int := 3;   // Rack Discharge State
      eRackMode_Circulate : Int := 4;   // Rack Circulate State
      eISEMode_Off : Int := 0;   // Skip dosing for this rack
      eISEMode_Load : Int := 1;   // Dose nutrients up to ISE High SP
      eISEMode_Deplete : Int := 2;   // Does nutrients up to ISE Low SP
   END_VAR


BEGIN
	// Rack Level Fertigation Controller
	// Responsible for: sending mutex lock requests to room, managing shelf valve and rack pump, and controlling rack state
	// Rack States:
	//      0 - Off
	//      1 - Fill
	//      2 - Measurement and Dosing
	//      3 - Discharge
	//      4 - Circulate (Default State)
	
	
	
	
	REGION 0: Off
	    // In the off state, close the shelf solenoid and turn off the pump
	    IF #Status.iState = #eRackMode_Off  THEN
	        #iOutMutexRequest := #eRackMode_Off;
	    END_IF;
	    
	    // wait to turn off shelf solenoid until pump stops
	    IF #Status.iState = #eRackMode_Off AND #Pump.Status.rActualSpeed = 0 THEN
	        #bShelfSolenoidCommand := 0;
	    END_IF;
	    
	END_REGION
	
	REGION 1: Fill
	    // In the fill state, send the mutex lock request, wait for confirmation, run the pump and open the shelf solenoid
	    // once the mutex lock drops out, move directly to 4: Circulate and set commanded mode to Circulate
	    
	    IF #Status.iState = #eRackMode_Fill THEN
	        
	        IF (#iInMutexLockConfirmation <> #eRackMode_Fill) AND NOT #bLockConfirmedModeActive THEN
	            #iOutMutexRequest := #eRackMode_Fill;
	        ELSIF #iInMutexLockConfirmation = #eRackMode_Fill THEN
	            #bLockConfirmedModeActive := 1;
	            #iOutMutexRequest := #eRackMode_Off;
	            #bShelfSolenoidCommand := 1;
	        ELSIF (#iInMutexLockConfirmation <> #eRackMode_Fill) AND #bLockConfirmedModeActive THEN
	            #bLockConfirmedModeActive := 0;
	            #iNextMode := #eRackMode_Circulate;
	            #Controls.iModeCommand := #eRackMode_Circulate;
	        END_IF;
	    END_IF;
	    
	    
	END_REGION
	
	REGION 2: Measurement & Dosing
	    // In the measurement and dosing state, send the mutex lock request along with the nutrient
	    // dosing setpoints, wait for confirmation, then automatically transition TO 4: Circulation
	        
	    IF #Status.iState = #eRackMode_MeasurementDosing THEN
	        
	        // request M&D lock
	        IF (#iInMutexLockConfirmation <> #eRackMode_MeasurementDosing) AND NOT #bLockConfirmedModeActive THEN
	            #iOutMutexRequest := #eRackMode_MeasurementDosing;
	            
	            // confirm that we are locked
	        ELSIF #iInMutexLockConfirmation = #eRackMode_MeasurementDosing AND NOT #bLockConfirmedModeActive THEN
	            #bLockConfirmedModeActive := 1;
	            #iOutMutexRequest := #eRackMode_Off;
	            #bShelfSolenoidCommand := 1;
	            #rInitialVolume := #rInReservoirLevel;
	            
	            // check that M&D is done, go back to circulate
	        ELSIF #iInMutexLockConfirmation <> #eRackMode_MeasurementDosing AND #bLockConfirmedModeActive THEN
	            #bLockConfirmedModeActive := 0;
	            #iNextMode := #eRackMode_Circulate;
	            #retVal := RD_LOC_T(#Controls.dtLastMeasurement); // save last time measurement has occured
	        END_IF;
	            
	    END_IF;
	    
	    
	END_REGION
	
	REGION 3: Discharge
	    // In the discharge state, send the mutex lock request, wait for confirmation, close shelf solenoid
	    // once the mutex lock drops out, move directly to 0: Off and set commanded mode to Off
	    
	    IF #Status.iState = #eRackMode_Discharge THEN
	        IF (#iInMutexLockConfirmation <> #eRackMode_Discharge) AND NOT #bLockConfirmedModeActive THEN
	            #iOutMutexRequest := #eRackMode_Discharge;
	        ELSIF #iInMutexLockConfirmation = #eRackMode_Discharge THEN
	            #bLockConfirmedModeActive := 1;
	            #iOutMutexRequest := #eRackMode_Off;
	            #bShelfSolenoidCommand := 0;
	        ELSIF (#iInMutexLockConfirmation <> #eRackMode_Discharge) AND #bLockConfirmedModeActive THEN
	            #bLockConfirmedModeActive := 0;
	            #iNextMode := #eRackMode_Off;
	            #Controls.iModeCommand := #eRackMode_Off;
	        END_IF;
	    ELSE
	        #Controls.bEndDischargeCommand := FALSE;
	    END_IF;
	    
	    #OutFertigationSettings.tDischargeTime := DINT_TO_TIME(#Controls.diDischargeTimeSecs * 1000);
	    #OutFertigationSettings.bEndDischargeCommand := #Controls.bEndDischargeCommand;
	    
	END_REGION
	
	REGION 4: Circulate
	    // In the circulate state, open the shelf solenoid and run the pump
	    // Mutex request to Room is off
	    IF #Status.iState = #eRackMode_Circulate THEN
	        #bShelfSolenoidCommand := 1;
	        #iOutMutexRequest := #eRackMode_Off;
	    END_IF;
	    
	    // Automatically trigger M&D after 2 hours of circulating if the commanded state is M&D
	    // 
	    #retVal := RD_LOC_T(OUT => #tCurrentDateTime);
	    
	    #lastDelta := T_SUB(IN1:=#tCurrentDateTime,
	                        IN2:=DINT_TO_TIME(#Controls.diDosingIntervalMins * 60 * 1000));
	    
	    IF (#Status.iState = #eRackMode_Circulate AND
	        #Controls.iModeCommand = #eRackMode_MeasurementDosing AND
	        #lastDelta > #Controls.dtLastMeasurement) THEN
	        #iNextMode := #eRackMode_MeasurementDosing;
	    END_IF;
	    
	    
	    (*
	    #TON_Circulate(IN := #Status.iState = #eRackMode_Circulate AND #Controls.iModeCommand = #eRackMode_MeasurementDosing,
	                   PT := DINT_TO_TIME(#Controls.diDosingIntervalMins * 60 * 1000));
	    
	    IF #TON_Circulate.Q THEN
	        #iNextMode := #eRackMode_MeasurementDosing;
	    END_IF;
	    *)
	    
	END_REGION
	
	REGION State Management
	    // If rack is in Off or Circulate, take the OPC commanded state
	    // Except if commanding M&D, go into circulate first, then it will automatically go into M&D on the timer
	    // If rack is in M&D, Fill, or Discharge, wait for the automatic state transition
	    
	    IF #Status.iState = #eRackMode_Off  AND #Controls.iModeCommand = #eRackMode_MeasurementDosing THEN
	        #iNextMode := #eRackMode_Circulate;
	        
	    ELSIF #Status.iState = #eRackMode_Off OR 
	        (#Status.iState = #eRackMode_Circulate AND #Controls.iModeCommand <> #eRackMode_MeasurementDosing) THEN
	        #iNextMode := #Controls.iModeCommand;
	        
	    END_IF;
	
	    #Status.iState := #iNextMode;
	    
	END_REGION
	
	
	REGION Pump Management
	    
	    IF #rInReservoirLevel < #Controls.rPumpReservoirInterlockLevel OR #Status.iState = #eRackMode_Off THEN
	        // turn off pump if there's not enough water
	        #rPumpSpeed := 0;
	        
	    ELSIF #Status.iState = #eRackMode_MeasurementDosing AND #bInReturnSolenoidStatus = 1 THEN
	        // returning water to the main tank, check that the return solenoid is open
	        #rPumpSpeed := #Controls.rPumpReturnSpeed;
	        
	    ELSIF #Status.iState = #eRackMode_Discharge AND #bInReturnSolenoidStatus = 1 THEN
	        // discharging water from rack reservoir to sewer, check that the return solenoid is open
	        #rPumpSpeed := #Controls.rPumpDischargeSpeed;
	        
	    ELSIF  #bInShelfSolenoidStatus = 1 THEN
	        // circulate mode, fill mode, and all other state, double check the the shelf solenoid is open
	        #rPumpSpeed := #Controls.rPumpContinousSpeed;
	        
	    ELSE
	        #rPumpSpeed := 0;
	        
	    END_IF;
	    
	    #Pump(rInSpeedCommand := #rPumpSpeed);
	              
	END_REGION
	
	REGION Fertigation Settings
	    // Package up OPC Settings for fertigation to pass out to room
	    
	    #OutFertigationSettings.tMeasurementTime := DINT_TO_TIME(#Controls.diMeasurementSecs * 1000);
	    #OutFertigationSettings.rMeasurementVolume := #Controls.rMeasurementVolume;
	    #OutFertigationSettings.bNutrientAEnable := #Controls.bNutrientAEnable;
	    #OutFertigationSettings.bNutrientBEnable := #Controls.bNutrientBEnable;
	    #OutFertigationSettings.rISELowSP := #Controls.rISELowSP;
	    #OutFertigationSettings.rISEHighSP := #Controls.rISEHighSP;
	    #OutFertigationSettings.tNutrientDosingDuration := DINT_TO_TIME(#Controls.diNutrientDosingSecs * 1000);
	    
	    #OutFertigationSettings.rOperatingVolume := #Controls.rOperatingVolume;
	    #OutFertigationSettings.rTotalShelfVolume := #Controls.rTotalShelfVolume;
	    #OutFertigationSettings.rMaxReservoirVolume := #Controls.rMaxReservoirVolume;
	    #OutFertigationSettings.rMinReservoirVolume := #Controls.rPumpReservoirInterlockLevel;
	    #OutFertigationSettings.rRackCurrentVolume := #rInReservoirLevel;
	    
	    #OutFertigationSettings.bPumpAtStandstill := #Pump.Status.rActualSpeed = 0;
	    
	    // Enable incoming rotate from room if in M&D mode and current state is circulate
	    #OutFertigationSettings.bEnableIncomingRotate := #Status.iState = #eRackMode_Circulate
	    AND #Controls.iModeCommand = #eRackMode_MeasurementDosing;
	    
	END_REGION
	    
	    
	    REGION ISE Mode
	        // Determine if dosing is required based off of ISE reading, low/high setpoints, and commanded ISE mode
	        
	        // if in load mode and high SP is reached, switch to deplete
	        IF #Controls.iISEModeCommand = #eISEMode_Load AND #InLastNutrientReading.rISEReading >= #Controls.rISEHighSP THEN
	            #Controls.iISEModeCommand := #eISEMode_Deplete;
	        END_IF;
	        
	        // if in deplete mode and low SP is reached, switch to load
	        IF #Controls.iISEModeCommand = #eISEMode_Deplete AND #InLastNutrientReading.rISEReading <= #Controls.rISELowSP THEN
	            #Controls.iISEModeCommand := #eISEMode_Load;
	        END_IF;
	        
	        // Request dosing if in load mode, skip dosing if in deplete or off
	        #OutFertigationSettings.bDosingActive := (#Controls.iISEModeCommand = #eISEMode_Load);
	        
	    //Copy over nutrient levels to OPC status output when M&D lock drops out
	    #NutrientReadingReady(CLK:= (#iInMutexLockConfirmation = #eRackMode_MeasurementDosing));
	    IF #NutrientReadingReady.Q THEN
	        #Status.NutrientLevels := #InLastNutrientReading;
	    END_IF;
	    
	    
	END_REGION
	
	REGION Set digital outputs
	    #bOutShelfSolenoid :=  #bShelfSolenoidCommand;
	    
	END_REGION
	
	
	
	
	
END_FUNCTION_BLOCK

FUNCTION_BLOCK "fbRackPump"   // FB10, LAD
{ S7_Optimized_Access := 'TRUE' }
VERSION : 0.1
// Pump has 3 modes: Off, Priming, Running. 
// If the pump speed changes from zero to non-zero, start priming for the priming duration
// Once priming is complete, move to Pump running while the rack remains in Fill or Circulate
// stored: AutoNumber true, IsIECCheckEnabled false, IsRetainMemResEnabled false, MemoryReserve 100, SetENOAutomatically false, UDAEnableTagReadback false
   VAR_INPUT
      rInSpeedCommand { ExternalAccessible := 'False'; ExternalVisible := 'False'; ExternalWritable := 'False'} : Real;   // Commanded pump speed (%)
   END_VAR
   VAR RETAIN
      Controls { ExternalVisible := 'False'} : Struct
         rPrimeSpeed { ExternalVisible := 'False'} : Real := 100.0;   // Pump speed when priming (%)
         diPrimingSecs { ExternalVisible := 'False'} : DInt := 60;   // Duration of pump priming (seconds)
         bOverrideEnable { ExternalVisible := 'False'} : Bool;   // Sets pump speed to the override value
         rOverrideSpeed { ExternalVisible := 'False'} : Real;   // Manual override speed (%) Set to 0 to turn off.
      END_STRUCT;
      Status { ExternalVisible := 'False'; ExternalWritable := 'False'} : Struct
         iState { ExternalVisible := 'False'; ExternalWritable := 'False'} : Int;   // 0: Off, 1: Priming, 2:Running
         rCommandSpeed { ExternalAccessible := 'False'; ExternalVisible := 'False'; ExternalWritable := 'False'} : Real;   // Speed commanded to VFD (%)
         rActualSpeed { ExternalVisible := 'False'; ExternalWritable := 'False'} : Real;   // Speed reported from VFD (%)
         rVoltage { ExternalVisible := 'False'; ExternalWritable := 'False'} : Real;   // Vrms
         rCurrent { ExternalVisible := 'False'; ExternalWritable := 'False'} : Real;   // Arms
         rPower { ExternalVisible := 'False'; ExternalWritable := 'False'} : Real;   // kW
         rPowerFactor { ExternalVisible := 'False'; ExternalWritable := 'False'} : Real;
         bError { ExternalVisible := 'False'; ExternalWritable := 'False'} : Bool;
         ErrorDetail { ExternalVisible := 'False'; ExternalWritable := 'False'} : "udtError_VFD";
      END_STRUCT;
   END_VAR
   VAR
      fbVFD { ExternalAccessible := 'False'; ExternalVisible := 'False'; ExternalWritable := 'False'} : "fbVFD_GSeries";
      TON_Priming { ExternalAccessible := 'False'; ExternalVisible := 'False'; ExternalWritable := 'False'} : TON_TIME;
      dummyUdt { ExternalAccessible := 'False'; ExternalVisible := 'False'; ExternalWritable := 'False'} : "udtHMI_VFD_Control";   // Ignore
   END_VAR
   VAR_TEMP
      arrTelegramWords : Array[1..6] of Int;
      iRet : Int;
   END_VAR
   VAR CONSTANT
      eStateOff : Int := 0;
      eStatePriming : Int := 1;
      eStateRunning : Int := 2;
      cScalingFactor : Real := 16384.0;   // Full scale (100%) value of VFD parameters
   END_VAR
BEGIN

REGION Network 1 (SCL): Determine pump VFD command speed based on off/priming/run state
   IF #rInSpeedCommand <> 0 THEN
       // start out by priming, then switch to running
       IF #Status.iState = #eStateOff THEN
           #Status.iState := #eStatePriming;
       ELSIF #Status.iState = #eStatePriming AND #TON_Priming.Q THEN
           #Status.iState := #eStateRunning;
       END_IF;

   ELSE
       #Status.iState := #eStateOff;
   END_IF;

   #TON_Priming(IN := (#Status.iState = #eStatePriming),
                PT := DINT_TO_TIME(#Controls.diPrimingSecs * 1000));

   // Check for manual override
   IF #Controls.bOverrideEnable THEN
       #fbVFD.rInCommandSpeed := #Controls.rOverrideSpeed;

   ELSE
       CASE #Status.iState OF
           #eStateOff: // Off
               #fbVFD.rInCommandSpeed := 0;
           #eStatePriming: // Priming - run at priming speed until priming timer has elapsed then transition to Running   
               #fbVFD.rInCommandSpeed := #Controls.rPrimeSpeed;
           #eStateRunning: // Running
               #fbVFD.rInCommandSpeed := #rInSpeedCommand;
       END_CASE;

       // if override is not active, override speed tracks command speed so that activating override mode
       // doesn't unexpectedly change the value
       #Controls.rOverrideSpeed := #fbVFD.rInCommandSpeed;

   END_IF;

   #Status.rCommandSpeed := #fbVFD.rInCommandSpeed;
END_REGION

REGION Network 2: Open library G series VFD block call
   // Telegram is assigned globally in fbConfig.
   // Contactor output is fed back since we con't have a physical one.
   // Dummy Udt is needed even though we don't have an HMI faceplate.
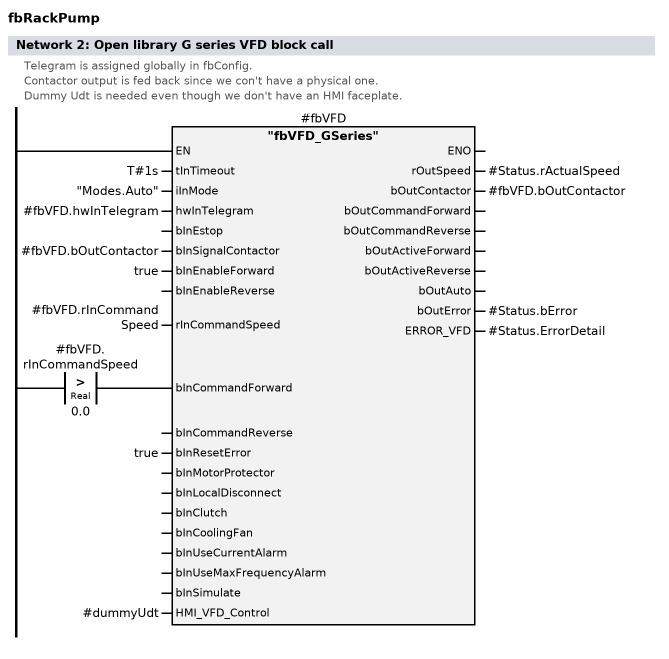
   RUNG wire#powerrail
      #fbVFD(bInCommandForward := wire#w1, tInTimeout := T#1s, iInMode := "Modes.Auto", hwInTelegram := #fbVFD.hwInTelegram, bInEstop :=, bInSignalContactor := #fbVFD.bOutContactor, bInEnableForward := true, bInEnableReverse :=, rInCommandSpeed := #fbVFD.rInCommandSpeed, bInCommandReverse :=, bInResetError := true, bInMotorProtector :=, bInLocalDisconnect :=, bInClutch :=, bInCoolingFan :=, bInUseCurrentAlarm :=, bInUseMaxFrequencyAlarm :=, bInSimulate :=, HMI_VFD_Control := #dummyUdt, rOutSpeed => #Status.rActualSpeed, bOutContactor => #fbVFD.bOutContactor, bOutCommandForward =>, bOutCommandReverse =>, bOutActiveForward =>, bOutActiveReverse =>, bOutAuto =>, bOutError => #Status.bError, ERROR_VFD => #Status.ErrorDetail)
   END_RUNG
   RUNG wire#powerrail
      { S7_Templates := "SrcType := Real" } GT_Contact(in1 := #fbVFD.rInCommandSpeed, in2 := 0.0)
   END_RUNG wire#w1
   // the same network as SCL:
   #fbVFD(tInTimeout := T#1s,   // "fbVFD_GSeries"
          iInMode := "Modes.Auto",
          hwInTelegram := #fbVFD.hwInTelegram,
          bInSignalContactor := #fbVFD.bOutContactor,
          bInEnableForward := true,
          rInCommandSpeed := #fbVFD.rInCommandSpeed,
          bInCommandForward := #fbVFD.rInCommandSpeed > 0.0,
          bInResetError := true,
          HMI_VFD_Control := #dummyUdt,
          rOutSpeed => #Status.rActualSpeed,
          bOutContactor => #fbVFD.bOutContactor,
          bOutError => #Status.bError,
          ERROR_VFD => #Status.ErrorDetail);
END_REGION

REGION Network 3 (SCL): Read additional drive parameters from exteneded telegram
   #iRet := DPRD_DAT(LADDR := #fbVFD.hwInTelegram, RECORD => #arrTelegramWords);

   // Telegram word 1 (status word) is handled inside fbVFD
   #Status.rActualSpeed := #arrTelegramWords[2] / #cScalingFactor * 100; // percent 
   #Status.rVoltage := #arrTelegramWords[3] / #cScalingFactor * 1000; // Vrms
   #Status.rCurrent := #arrTelegramWords[4] / #cScalingFactor * 7.1; //9.43; // Arms
   #Status.rPower := #arrTelegramWords[5] / #cScalingFactor * 1.49 * 2;//3.15; // Kw
   #Status.rPowerFactor := #arrTelegramWords[6] / #cScalingFactor;
END_REGION
END_FUNCTION_BLOCK

